	{attribute 'TcIecLibraryType'}
	{attribute 'external_name' := 'F_VN_ApplyYAxisInversionToAffineTransformationExp_GUID_95763161_5894_2E34_6A2A_637EF808A786'}
	(* Apply an inversion of the y-axis direction to an existing 2D affine transformation matrix. (expert function) *)
	FUNCTION F_VN_ApplyYAxisInversionToAffineTransformationExp : HRESULT
	VAR_IN_OUT
		aTransformationMatrix	:	TcVnMatrix2x3_LREAL;	(* Affine transformation matrix to which the inversion of the y-axis direction is applied *)
	END_VAR
	VAR_INPUT
		bUsePreMultiplication	:	BOOL;	(* Select if pre- or post-multiplication should be used *)
		hrPrev	:	HRESULT;	(* HRESULT indicating the result of previous operations (If SUCCEEDED(hrPrev) equals false, no operation is executed.) *)
	END_VAR

END_FUNCTION

// Functions/Geometric and Coordinate Transformations/F_VN_ConvertCartesianToPolarAngleImage

	{attribute 'TcIecLibraryType'}
	{attribute 'external_name' := 'F_VN_ConvertCartesianToPolarAngleImage_GUID_8785DF50_8290_2A16_55B0_D427D2D5A086'}
	(* Converts cartesian coordinates (x, y) to polar angle. *)
	FUNCTION F_VN_ConvertCartesianToPolarAngleImage : HRESULT
	VAR_INPUT
		ipSrcImageX	:	ITcVnImage;	(* Source image containing the x values (elements of type REAL or LREAL) *)
		ipSrcImageY	:	ITcVnImage;	(* Source image containing the y values (Same element type as ipSrcImageX) *)
		ipDestImageAng	:	REFERENCE TO ITcVnImage;	(* Destination image containing the angles (Same element type as source images. An appropriate destination image will be created if required.) *)
		hrPrev	:	HRESULT;	(* HRESULT indicating the result of previous operations (If SUCCEEDED(hrPrev) equals false, no operation is executed.) *)
	END_VAR

END_FUNCTION

// Functions/Geometric and Coordinate Transformations/F_VN_ConvertCartesianToPolarAngleImageExp

	{attribute 'TcIecLibraryType'}
	{attribute 'external_name' := 'F_VN_ConvertCartesianToPolarAngleImageExp_GUID_8D077096_5D1D_2FC1_51E8_F25300BF841D'}
	(* Converts cartesian coordinates (x, y) to polar angle. (expert function) *)
	FUNCTION F_VN_ConvertCartesianToPolarAngleImageExp : HRESULT
	VAR_INPUT
		ipSrcImageX	:	ITcVnImage;	(* Source image containing the x values (elements of type REAL or LREAL) *)
		ipSrcImageY	:	ITcVnImage;	(* Source image containing the y values (Same element type as ipSrcImageX) *)
		ipDestImageAng	:	REFERENCE TO ITcVnImage;	(* Destination image containing the angles (Same element type as source images. An appropriate destination image will be created if required.) *)
		bAngleInDegrees	:	BOOL;	(* Specifys, if the angles should be in degrees or radians *)
		hrPrev	:	HRESULT;	(* HRESULT indicating the result of previous operations (If SUCCEEDED(hrPrev) equals false, no operation is executed.) *)
	END_VAR

END_FUNCTION

// Functions/Geometric and Coordinate Transformations/F_VN_ConvertCartesianToPolarAngles

	{attribute 'TcIecLibraryType'}
	{attribute 'external_name' := 'F_VN_ConvertCartesianToPolarAngles_GUID_777B4F5A_64D8_2B5B_6D5A_3B670B4891DC'}
	(* Converts cartesian coordinates (x, y) to polar angle. *)
	FUNCTION F_VN_ConvertCartesianToPolarAngles : HRESULT
	VAR_INPUT
		ipSrcPointsCart	:	ITcVnContainer;	(* Container with cartesian points (ContainerType_Vector_TcVnPoint2_DINT or ContainerType_Vector_TcVnPoint2_REAL or ContainerType_Vector_TcVnPoint2_LREAL) *)
		ipDestAngles	:	REFERENCE TO ITcVnContainer;	(* Returns a container which is filled with the angles (ContainerType_Vector_REAL, if source points are of type TcVnPoint2_DINT or TcVnPoint2_REAL; else ContainerType_Vector_LREAL. Non-zero interface pointers are reused.) *)
		hrPrev	:	HRESULT;	(* HRESULT indicating the result of previous operations (If SUCCEEDED(hrPrev) equals false, no operation is executed.) *)
	END_VAR

END_FUNCTION

// Functions/Geometric and Coordinate Transformations/F_VN_ConvertCartesianToPolarAnglesExp

	{attribute 'TcIecLibraryType'}
	{attribute 'external_name' := 'F_VN_ConvertCartesianToPolarAnglesExp_GUID_C17BBC53_AA08_2C58_6EA5_EB565B2A30B9'}
	(* Converts cartesian coordinates (x, y) to polar angle. (expert function) *)
	FUNCTION F_VN_ConvertCartesianToPolarAnglesExp : HRESULT
	VAR_INPUT
		ipSrcPointsCart	:	ITcVnContainer;	(* Container with cartesian points (ContainerType_Vector_TcVnPoint2_DINT or ContainerType_Vector_TcVnPoint2_REAL or ContainerType_Vector_TcVnPoint2_LREAL) *)
		ipDestAngles	:	REFERENCE TO ITcVnContainer;	(* Returns a container which is filled with the angles (ContainerType_Vector_REAL, if source points are of type TcVnPoint2_DINT or TcVnPoint2_REAL; else ContainerType_Vector_LREAL. Non-zero interface pointers are reused.) *)
		bAngleInDegrees	:	BOOL;	(* Specify, if the angles should be in degrees or radians *)
		hrPrev	:	HRESULT;	(* HRESULT indicating the result of previous operations (If SUCCEEDED(hrPrev) equals false, no operation is executed.) *)
	END_VAR

END_FUNCTION

// Functions/Geometric and Coordinate Transformations/F_VN_ConvertCartesianToPolarImages

	{attribute 'TcIecLibraryType'}
	{attribute 'external_name' := 'F_VN_ConvertCartesianToPolarImages_GUID_68D50C9F_CB61_2D1C_5256_8997FCBD3F82'}
	(* Converts cartesian coordinates (x, y) to polar coordinates (magnitude, angle). *)
	FUNCTION F_VN_ConvertCartesianToPolarImages : HRESULT
	VAR_INPUT
		ipSrcImageX	:	ITcVnImage;	(* Source image containing the x values (elements of type REAL or LREAL) *)
		ipSrcImageY	:	ITcVnImage;	(* Source image containing the y values (Same element type as ipSrcImageX) *)
		ipDestImageMag	:	REFERENCE TO ITcVnImage;	(* Destination image containing the magnitudes (Same element type as source images. An appropriate destination image will be created if required.) *)
		ipDestImageAng	:	REFERENCE TO ITcVnImage;	(* Destination image containing the angles (Same element type as source images. An appropriate destination image will be created if required.) *)
		hrPrev	:	HRESULT;	(* HRESULT indicating the result of previous operations (If SUCCEEDED(hrPrev) equals false, no operation is executed.) *)
	END_VAR

END_FUNCTION

// Functions/Geometric and Coordinate Transformations/F_VN_ConvertCartesianToPolarImagesExp

	{attribute 'TcIecLibraryType'}
	{attribute 'external_name' := 'F_VN_ConvertCartesianToPolarImagesExp_GUID_57A46AC2_A055_2CB3_451E_4402032FA64B'}
	(* Converts cartesian coordinates (x, y) to polar coordinates (magnitude, angle). (expert function) *)
	FUNCTION F_VN_ConvertCartesianToPolarImagesExp : HRESULT
	VAR_INPUT
		ipSrcImageX	:	ITcVnImage;	(* Source image containing the x values (elements of type REAL or LREAL) *)
		ipSrcImageY	:	ITcVnImage;	(* Source image containing the y values (Same element type as ipSrcImageX) *)
		ipDestImageMag	:	REFERENCE TO ITcVnImage;	(* Destination image containing the magnitudes (Same element type as source images. An appropriate destination image will be created if required.) *)
		ipDestImageAng	:	REFERENCE TO ITcVnImage;	(* Destination image containing the angles (Same element type as source images. An appropriate destination image will be created if required.) *)
		bAngleInDegrees	:	BOOL;	(* Specifys, if the angles should be in degrees or radians *)
		hrPrev	:	HRESULT;	(* HRESULT indicating the result of previous operations (If SUCCEEDED(hrPrev) equals false, no operation is executed.) *)
	END_VAR

END_FUNCTION

// Functions/Geometric and Coordinate Transformations/F_VN_ConvertCartesianToPolarMagnitudeImage

	{attribute 'TcIecLibraryType'}
	{attribute 'external_name' := 'F_VN_ConvertCartesianToPolarMagnitudeImage_GUID_99EFD0C0_CF11_2C59_5201_85CBDF72A9FC'}
	(* Converts cartesian coordinates (x, y) to polar magnitude. *)
	FUNCTION F_VN_ConvertCartesianToPolarMagnitudeImage : HRESULT
	VAR_INPUT
		ipSrcImageX	:	ITcVnImage;	(* Source image containing the x values (elements of type REAL or LREAL) *)
		ipSrcImageY	:	ITcVnImage;	(* Source image containing the y values (Same element type as ipSrcImageX) *)
		ipDestImageMag	:	REFERENCE TO ITcVnImage;	(* Destination image containing the magnitudes (Same element type as source images. An appropriate destination image will be created if required.) *)
		hrPrev	:	HRESULT;	(* HRESULT indicating the result of previous operations (If SUCCEEDED(hrPrev) equals false, no operation is executed.) *)
	END_VAR

END_FUNCTION

// Functions/Geometric and Coordinate Transformations/F_VN_ConvertCartesianToPolarMagnitudes

	{attribute 'TcIecLibraryType'}
	{attribute 'external_name' := 'F_VN_ConvertCartesianToPolarMagnitudes_GUID_87575312_399C_21BE_5CEE_FFE66CC03CE2'}
	(* Converts cartesian coordinates (x, y) to polar magnitude. *)
	FUNCTION F_VN_ConvertCartesianToPolarMagnitudes : HRESULT
	VAR_INPUT
		ipSrcPointsCart	:	ITcVnContainer;	(* Container with cartesian points (ContainerType_Vector_TcVnPoint2_DINT or ContainerType_Vector_TcVnPoint2_REAL or ContainerType_Vector_TcVnPoint2_LREAL) *)
		ipDestMags	:	REFERENCE TO ITcVnContainer;	(* Returns a container which is filled with the magnitudes (ContainerType_Vector_REAL, if source points are of type TcVnPoint2_DINT or TcVnPoint2_REAL; else ContainerType_Vector_LREAL. Non-zero interface pointers are reused.) *)
		hrPrev	:	HRESULT;	(* HRESULT indicating the result of previous operations (If SUCCEEDED(hrPrev) equals false, no operation is executed.) *)
	END_VAR

END_FUNCTION

// Functions/Geometric and Coordinate Transformations/F_VN_ConvertCartesianToPolarPoints

	{attribute 'TcIecLibraryType'}
	{attribute 'external_name' := 'F_VN_ConvertCartesianToPolarPoints_GUID_8B11E781_4477_2A78_64E3_1080D7128B46'}
	(* Converts cartesian coordinates (x, y) to polar coordinates (magnitude, angle). *)
	FUNCTION F_VN_ConvertCartesianToPolarPoints : HRESULT
	VAR_INPUT
		ipSrcPointsCart	:	ITcVnContainer;	(* Container with cartesian points (ContainerType_Vector_TcVnPoint2_DINT or ContainerType_Vector_TcVnPoint2_REAL or ContainerType_Vector_TcVnPoint2_LREAL) *)
		ipDestPointsPolar	:	REFERENCE TO ITcVnContainer;	(* Returns a container which is filled with the converted points in polar coordinates (ContainerType_Vector_TcVnPoint2_REAL, if source points are of type TcVnPoint2_DINT or TcVnPoint2_REAL; else ContainerType_Vector_TcVnPoint2_LREAL. Non-zero interface pointers are reused.) *)
		hrPrev	:	HRESULT;	(* HRESULT indicating the result of previous operations (If SUCCEEDED(hrPrev) equals false, no operation is executed.) *)
	END_VAR

END_FUNCTION

// Functions/Geometric and Coordinate Transformations/F_VN_ConvertCartesianToPolarPointsExp

	{attribute 'TcIecLibraryType'}
	{attribute 'external_name' := 'F_VN_ConvertCartesianToPolarPointsExp_GUID_EBBE416A_22C1_27E0_4531_5F2A0458D967'}
	(* Converts cartesian coordinates (x, y) to polar coordinates (magnitude, angle). (expert function) *)
	FUNCTION F_VN_ConvertCartesianToPolarPointsExp : HRESULT
	VAR_INPUT
		ipSrcPointsCart	:	ITcVnContainer;	(* Container with cartesian points (ContainerType_Vector_TcVnPoint2_DINT or ContainerType_Vector_TcVnPoint2_REAL or ContainerType_Vector_TcVnPoint2_LREAL) *)
		ipDestPointsPolar	:	REFERENCE TO ITcVnContainer;	(* Returns a container which is filled with the converted points in polar coordinates (ContainerType_Vector_TcVnPoint2_REAL, if source points are of type TcVnPoint2_DINT or TcVnPoint2_REAL; else ContainerType_Vector_TcVnPoint2_LREAL. Non-zero interface pointers are reused.) *)
		bAngleInDegrees	:	BOOL;	(* Specifys, if the angles should be in degrees or radians *)
		hrPrev	:	HRESULT;	(* HRESULT indicating the result of previous operations (If SUCCEEDED(hrPrev) equals false, no operation is executed.) *)
	END_VAR

END_FUNCTION

// Functions/Geometric and Coordinate Transformations/F_VN_ConvertPolarToCartesianImages

	{attribute 'TcIecLibraryType'}
	{attribute 'external_name' := 'F_VN_ConvertPolarToCartesianImages_GUID_45E29034_812A_29F4_4EDE_5DEB6A02A42A'}
	(* Converts polar coordinates (magnitude, angle) to cartesian coordinates (x, y). *)
	FUNCTION F_VN_ConvertPolarToCartesianImages : HRESULT
	VAR_INPUT
		ipSrcImageMag	:	ITcVnImage;	(* Source image containing the magnitudes (elements of type REAL or LREAL) *)
		ipSrcImageAng	:	ITcVnImage;	(* Source image containing the angles (Same element type as ipSrcImageMag) *)
		ipDestImageX	:	REFERENCE TO ITcVnImage;	(* Destination image containing the x values (Same element type as source images. An appropriate destination image will be created if required.) *)
		ipDestImageY	:	REFERENCE TO ITcVnImage;	(* Destination image containing the y values (Same element type as source images. An appropriate destination image will be created if required.) *)
		hrPrev	:	HRESULT;	(* HRESULT indicating the result of previous operations (If SUCCEEDED(hrPrev) equals false, no operation is executed.) *)
	END_VAR

END_FUNCTION

// Functions/Geometric and Coordinate Transformations/F_VN_ConvertPolarToCartesianImagesExp

	{attribute 'TcIecLibraryType'}
	{attribute 'external_name' := 'F_VN_ConvertPolarToCartesianImagesExp_GUID_1AB5C748_33A4_22CB_7CB8_EEAC3F1ECB67'}
	(* Converts polar coordinates (magnitude, angle) to cartesian coordinates (x, y). (expert function) *)
	FUNCTION F_VN_ConvertPolarToCartesianImagesExp : HRESULT
	VAR_INPUT
		ipSrcImageMag	:	ITcVnImage;	(* Source image containing the magnitudes (elements of type REAL or LREAL) *)
		ipSrcImageAng	:	ITcVnImage;	(* Source image containing the angles (Same element type as ipSrcImageMag) *)
		ipDestImageX	:	REFERENCE TO ITcVnImage;	(* Destination image containing the x values (Same element type as source images. An appropriate destination image will be created if required.) *)
		ipDestImageY	:	REFERENCE TO ITcVnImage;	(* Destination image containing the y values (Same element type as source images. An appropriate destination image will be created if required.) *)
		bAngleInDegrees	:	BOOL;	(* Specifys, if the angles are in degrees or radians *)
		hrPrev	:	HRESULT;	(* HRESULT indicating the result of previous operations (If SUCCEEDED(hrPrev) equals false, no operation is executed.) *)
	END_VAR

END_FUNCTION

// Functions/Geometric and Coordinate Transformations/F_VN_ConvertPolarToCartesianPoints

	{attribute 'TcIecLibraryType'}
	{attribute 'external_name' := 'F_VN_ConvertPolarToCartesianPoints_GUID_CD991F11_BA52_23B9_7986_18C4D3FB967A'}
	(* Converts polar coordinates (magnitude, angle) to cartesian coordinates (x, y). *)
	FUNCTION F_VN_ConvertPolarToCartesianPoints : HRESULT
	VAR_INPUT
		ipSrcPointsPolar	:	ITcVnContainer;	(* Container with polar coordinates (ContainerType_Vector_TcVnPoint2_REAL or ContainerType_Vector_TcVnPoint2_LREAL) *)
		ipDestPointsCart	:	REFERENCE TO ITcVnContainer;	(* Returns a container which is filled with the converted points in cartesian coordinates (same type ID as ipSrcPointsPolar. Non-zero interface pointers are reused.) *)
		hrPrev	:	HRESULT;	(* HRESULT indicating the result of previous operations (If SUCCEEDED(hrPrev) equals false, no operation is executed.) *)
	END_VAR

END_FUNCTION

// Functions/Geometric and Coordinate Transformations/F_VN_ConvertPolarToCartesianPointsExp

	{attribute 'TcIecLibraryType'}
	{attribute 'external_name' := 'F_VN_ConvertPolarToCartesianPointsExp_GUID_918F4026_8031_2284_7371_9471AA009DB3'}
	(* Converts polar coordinates (magnitude, angle) to cartesian coordinates (x, y). (expert function) *)
	FUNCTION F_VN_ConvertPolarToCartesianPointsExp : HRESULT
	VAR_INPUT
		ipSrcPointsPolar	:	ITcVnContainer;	(* Container with polar coordinates (ContainerType_Vector_TcVnPoint2_REAL or ContainerType_Vector_TcVnPoint2_LREAL) *)
		ipDestPointsCart	:	REFERENCE TO ITcVnContainer;	(* Returns a container which is filled with the converted points in cartesian coordinates (same type ID as ipSrcPointsPolar. Non-zero interface pointers are reused.) *)
		bAngleInDegrees	:	BOOL;	(* Specifys, if the angles are in degrees or radians *)
		hrPrev	:	HRESULT;	(* HRESULT indicating the result of previous operations (If SUCCEEDED(hrPrev) equals false, no operation is executed.) *)
	END_VAR

END_FUNCTION

// Functions/Geometric and Coordinate Transformations/F_VN_DecomposeAffineTransformation

	{attribute 'TcIecLibraryType'}
	{attribute 'external_name' := 'F_VN_DecomposeAffineTransformation_GUID_98D5C342_86DD_2C0D_79C0_D5DCC34233C1'}
	(* Decompose an affine transformation matrix and return the rotation angle (clockwise) in radian. The decomposition method assumes the following order of transformation: Translation, Rotation, Scale, and Skew. *)
	FUNCTION F_VN_DecomposeAffineTransformation : HRESULT
	VAR_IN_OUT
		aAffineTransform	:	TcVnMatrix2x3_LREAL;	(* Affine transformation matrix *)
		fRotationAngle	:	LREAL;	(* Rotation angle (radian) in the clockwise direction. The rotation center is the origin point (0,0) *)
	END_VAR
	VAR_INPUT
		hrPrev	:	HRESULT;	(* HRESULT indicating the result of previous operations (If SUCCEEDED(hrPrev) equals false, no operation is executed.) *)
	END_VAR

END_FUNCTION

// Functions/Geometric and Coordinate Transformations/F_VN_DecomposeAffineTransformationExp

	{attribute 'TcIecLibraryType'}
	{attribute 'external_name' := 'F_VN_DecomposeAffineTransformationExp_GUID_9A76BFDE_9FD8_208E_5443_0689F70E8650'}
	(* Decompose an affine transformation matrix and return the rotation angle (clockwise) in radian, translation vector (pixels), scale, and skew vectors (angle in radian). The decomposition method assumes the following order of transformation: Translation, Rotation, Scale, and Skew. *)
	FUNCTION F_VN_DecomposeAffineTransformationExp : HRESULT
	VAR_IN_OUT
		aAffineTransform	:	TcVnMatrix2x3_LREAL;	(* Affine transformation matrix *)
		fRotationAngle	:	LREAL;	(* Rotation angle (radian) in the clockwise direction. The rotation center is the origin point (0,0) *)
		aTranslationVector	:	TcVnVector2_LREAL;	(* 2D translation vector. The values are in pixels *)
		aScaleVector	:	TcVnVector2_LREAL;	(* 2D scale vector  *)
		aSkewVector	:	TcVnVector2_LREAL;	(* 2D skew vector. The values are the skew angles in x and y directions in radian *)
	END_VAR
	VAR_INPUT
		hrPrev	:	HRESULT;	(* HRESULT indicating the result of previous operations (If SUCCEEDED(hrPrev) equals false, no operation is executed.) *)
	END_VAR

END_FUNCTION

// Functions/Geometric and Coordinate Transformations/F_VN_DecomposeHomography

	{attribute 'TcIecLibraryType'}
	{attribute 'external_name' := 'F_VN_DecomposeHomography_GUID_98F01A4A_1DBD_2075_5784_A350D33354E2'}
	(* Decompose a homography matrix into four solutions of rotation, translation, and plane normal. It returns two solutions (Ra, Ta, Nb) and (Rb, Tb, Nb). The third and the fourth solutions can be calculated as follows: (Ra, -Ta, -Na) and (Rb, -Tb, -Nb). *)
	FUNCTION F_VN_DecomposeHomography : HRESULT
	VAR_IN_OUT
		aHomography	:	TcVnMatrix3x3_LREAL;	(* Homography matrix (a perspective transformation between two planes) *)
		aCameraMatrix	:	TcVnMatrix3x3_LREAL;	(* Camera matrix *)
		aRotationMatrixA	:	TcVnMatrix3x3_LREAL;	(* Rotation matrix of the first solution (Ra) *)
		aTranslationVectorA	:	TcVnVector3_LREAL;	(* Translation vector of the first solution (Ta) *)
		aNormVectorA	:	TcVnVector3_LREAL;	(* Norm vector of the first solution (Na) *)
		aRotationMatrixB	:	TcVnMatrix3x3_LREAL;	(* Rotation matrix of the second solution (Rb) *)
		aTranslationVectorB	:	TcVnVector3_LREAL;	(* Translation vector of the second solution (Tb) *)
		aNormVectorB	:	TcVnVector3_LREAL;	(* Norm vector of the second solution Nb *)
	END_VAR
	VAR_INPUT
		hrPrev	:	HRESULT;	(* HRESULT indicating the result of previous operations (If SUCCEEDED(hrPrev) equals false, no operation is executed.) *)
	END_VAR
	VAR_OUTPUT
		nSolutions	:	UDINT;	(* Returns the number of solutions. In normal cases, it is equal four.  *)
	END_VAR

END_FUNCTION

// Functions/Geometric and Coordinate Transformations/F_VN_DecomposeHomographyExp

	{attribute 'TcIecLibraryType'}
	{attribute 'external_name' := 'F_VN_DecomposeHomographyExp_GUID_E4534782_F1E5_2C71_56D0_408A9351CD4C'}
	(* Decompose a homography matrix and verify four solutions of rotation, translation, and plane normal. It uses visible reference points being in front of the camera to confirm which solution(s) of the four solutions (maximum two solutions) are consistent with all reference points. *)
	FUNCTION F_VN_DecomposeHomographyExp : HRESULT
	VAR_IN_OUT
		aHomography	:	TcVnMatrix3x3_LREAL;	(* Homography matrix (a perspective transformation between two planes) *)
		aCameraMatrix	:	TcVnMatrix3x3_LREAL;	(* Camera matrix *)
		aRotationMatrixA	:	TcVnMatrix3x3_LREAL;	(* Rotation matrix of the first solution (Ra) *)
		aTranslationVectorA	:	TcVnVector3_LREAL;	(* Translation vector of the first solution (Ta) *)
		aNormVectorA	:	TcVnVector3_LREAL;	(* Norm vector of the first solution (Na) *)
		aRotationMatrixB	:	TcVnMatrix3x3_LREAL;	(* Rotation matrix of the second solution (Rb) *)
		aTranslationVectorB	:	TcVnVector3_LREAL;	(* Translation vector of the second solution (Tb) *)
		aNormVectorB	:	TcVnVector3_LREAL;	(* Norm vector of the second solution (Nb) *)
	END_VAR
	VAR_INPUT
		ipPointsSrc	:	ITcVnContainer;	(* Container with source points (ContainerType_Vector_TcVnPoint2_REAL) *)
		ipPointsDes	:	ITcVnContainer;	(* Container with destination points (same number as ipPoints1, ContainerType_Vector_TcVnPoint2_REAL) *)
		ipInlierMask	:	ITcVnContainer;	(* A mask marking the inliers (optional, set to 0 if not available; ContainerType_Vector_SINT or ContainerType_Vector_USINT) *)
		hrPrev	:	HRESULT;	(* HRESULT indicating the result of previous operations (If SUCCEEDED(hrPrev) equals false, no operation is executed.) *)
	END_VAR
	VAR_OUTPUT
		nSolutions	:	UDINT;	(* Return the number of true potential solutions [0,1, or 2].
							0: no true potential solutions for the given corresponding points are confirmed.
							1: the solution (Ra, Ta, Na) is confirmed.
							2: both solution (Ra, Ta, Na) and (Rb, Tb, Nb) are confirmed.
							In all cases the function returns two solutions (Ra, Ta, Nb) and (Rb, Tb, Nb). The third and the fourth solutions can be calculated as follows: (Ra, -Ta, -Na) and (Rb, -Tb, -Nb).
						 *)
	END_VAR

END_FUNCTION

// Functions/Geometric and Coordinate Transformations/F_VN_FlipImage

	{attribute 'TcIecLibraryType'}
	{attribute 'external_name' := 'F_VN_FlipImage_GUID_48B32E72_66CF_244B_574F_84B8CCCB3BE5'}
	(* Flip an image (mirror and shift back to prior coordinates). *)
	FUNCTION F_VN_FlipImage : HRESULT
	VAR_INPUT
		ipSrcImage	:	ITcVnImage;	(* Source image *)
		ipDestImage	:	REFERENCE TO ITcVnImage;	(* Destination image (An appropriate destination image will be created if required.) *)
		eFlipAxis	:	ETcVnFlipAxis;	(* Selects the axis around which to flip the image *)
		hrPrev	:	HRESULT;	(* HRESULT indicating the result of previous operations (If SUCCEEDED(hrPrev) equals false, no operation is executed.) *)
	END_VAR

END_FUNCTION

// Functions/Geometric and Coordinate Transformations/F_VN_GenerateAffineTransformationUnitMatrix2D

	{attribute 'TcIecLibraryType'}
	{attribute 'external_name' := 'F_VN_GenerateAffineTransformationUnitMatrix2D_GUID_0E766047_45D3_2A7A_5039_15231E2195FF'}
	(* Generate an affine transformation 2D unit matrix. *)
	FUNCTION F_VN_GenerateAffineTransformationUnitMatrix2D : HRESULT
	VAR_IN_OUT
		aTransformationMatrix	:	TcVnMatrix2x3_LREAL;	(* Resulting affine transformation unit matrix *)
	END_VAR
	VAR_INPUT
		hrPrev	:	HRESULT;	(* HRESULT indicating the result of previous operations (If SUCCEEDED(hrPrev) equals false, no operation is executed.) *)
	END_VAR

END_FUNCTION

// Functions/Geometric and Coordinate Transformations/F_VN_GetAffineTransformation

	{attribute 'TcIecLibraryType'}
	{attribute 'external_name' := 'F_VN_GetAffineTransformation_GUID_7F9475AC_C0C6_2ED5_5448_BF3DBD7E8953'}
	(* Calculate the affine transformation between three corresponding point pairs. The points mark the corners of the corresponding triangles. *)
	FUNCTION F_VN_GetAffineTransformation : HRESULT
	VAR_IN_OUT
		aSrcPoints	:	TcVnArray3_Point2_REAL;	(* Source points *)
		aDestPoints	:	TcVnArray3_Point2_REAL;	(* Destination points *)
		aTransformationMatrix	:	TcVnMatrix2x3_LREAL;	(* Resulting transformation matrix *)
	END_VAR
	VAR_INPUT
		hrPrev	:	HRESULT;	(* HRESULT indicating the result of previous operations (If SUCCEEDED(hrPrev) equals false, no operation is executed.) *)
	END_VAR

END_FUNCTION

// Functions/Geometric and Coordinate Transformations/F_VN_GetAffineTransformation2D

	{attribute 'TcIecLibraryType'}
	{attribute 'external_name' := 'F_VN_GetAffineTransformation2D_GUID_75CFB795_4F15_2741_5A15_1A9F0AAB074F'}
	(* Estimate the 2D affine transformation between two planar point sets using RANSAC algorithm. *)
	FUNCTION F_VN_GetAffineTransformation2D : HRESULT
	VAR_INPUT
		ipSrcPoints	:	ITcVnContainer;	(* Container with at least 3 source points (ContainerType_Vector_TcVnPoint2_REAL) *)
		ipDestPoints	:	ITcVnContainer;	(* Container with destination points (same number as ipSrcPoints, ContainerType_Vector_TcVnPoint2_REAL) *)
	END_VAR
	VAR_IN_OUT
		aAffineTransform	:	TcVnMatrix2x3_LREAL;	(* Returns the affine transformation matrix, which transforms the source points to the destination points *)
	END_VAR
	VAR_INPUT
		hrPrev	:	HRESULT;	(* HRESULT indicating the result of previous operations (If SUCCEEDED(hrPrev) equals false, no operation is executed.) *)
	END_VAR

END_FUNCTION

// Functions/Geometric and Coordinate Transformations/F_VN_GetAffineTransformation2DExp

	{attribute 'TcIecLibraryType'}
	{attribute 'external_name' := 'F_VN_GetAffineTransformation2DExp_GUID_A72EB0C5_44D0_245E_5406_EFAD4AF3D8CC'}
	(* Estimate the affine transformation between two planar point sets. (expert function) *)
	FUNCTION F_VN_GetAffineTransformation2DExp : HRESULT
	VAR_INPUT
		ipSrcPoints	:	ITcVnContainer;	(* Container with at least 3 source points (ContainerType_Vector_TcVnPoint2_REAL) *)
		ipDestPoints	:	ITcVnContainer;	(* Container with destination points (same number as ipSrcPoints, ContainerType_Vector_TcVnPoint2_REAL) *)
	END_VAR
	VAR_IN_OUT
		aAffineTransform	:	TcVnMatrix2x3_LREAL;	(* Returns the affine transformation matrix, which transforms the source points to the destination points *)
	END_VAR
	VAR_INPUT
		eAlgorithm	:	ETcVnEstimationAlgorithm;	(* Estimation algorithm (only RANSAC and LMEDS are supported) *)
		fReprojThreshold	:	LREAL;	(* Maximum allowed reprojection error to treat a point pair as an inlier *)
		ipInlierMask	:	REFERENCE TO ITcVnContainer;	(* Returns a mask marking the inliers (optional, set to 0 if not required; ContainerType_Vector_USINT) *)
		nMaxIterations	:	UDINT;	(* Maximum number of iterations *)
		fConfidence	:	LREAL;	(* Confidence (0..1) *)
		nRefineIters	:	UDINT;	(* Maximum number of iterations of Levenberg-Marquardt algorithm to refine further the affine transform (using only inliers). Set to 0 to disable refining. *)
		hrPrev	:	HRESULT;	(* HRESULT indicating the result of previous operations (If SUCCEEDED(hrPrev) equals false, no operation is executed.) *)
	END_VAR

END_FUNCTION

// Functions/Geometric and Coordinate Transformations/F_VN_GetPerspectiveTransformation

	{attribute 'TcIecLibraryType'}
	{attribute 'external_name' := 'F_VN_GetPerspectiveTransformation_GUID_F37A28EB_B072_2EC2_73AC_6B19B9A31E9E'}
	(* Calculate the perspective transformation between four corresponding point pairs. The points mark the corners of the corresponding rectangles. *)
	FUNCTION F_VN_GetPerspectiveTransformation : HRESULT
	VAR_IN_OUT
		aSrcPoints	:	TcVnArray4_Point2_REAL;	(* Source points *)
		aDestPoints	:	TcVnArray4_Point2_REAL;	(* Destination points *)
		aTransformationMatrix	:	TcVnMatrix3x3_LREAL;	(* Resulting transformation matrix *)
	END_VAR
	VAR_INPUT
		hrPrev	:	HRESULT;	(* HRESULT indicating the result of previous operations (If SUCCEEDED(hrPrev) equals false, no operation is executed.) *)
	END_VAR

END_FUNCTION

// Functions/Geometric and Coordinate Transformations/F_VN_Homography

	{attribute 'TcIecLibraryType'}
	{attribute 'external_name' := 'F_VN_Homography_GUID_8DBA4BBF_8913_20A2_43C2_DD73C62F3751'}
	(* Find the homography (perspective transformation) between two planar point sets using RANSAC algorithm. *)
	FUNCTION F_VN_Homography : HRESULT
	VAR_INPUT
		ipSrcPoints	:	ITcVnContainer;	(* Container with at least 4 source points (ContainerType_Vector_TcVnPoint2_REAL) *)
		ipDestPoints	:	ITcVnContainer;	(* Container with destination points (same number as ipSrcPoints, ContainerType_Vector_TcVnPoint2_REAL) *)
	END_VAR
	VAR_IN_OUT
		aPerspectiveTransform	:	TcVnMatrix3x3_LREAL;	(* Returns the perspective transformation matrix, which transforms the source points to the destination points *)
	END_VAR
	VAR_INPUT
		hrPrev	:	HRESULT;	(* HRESULT indicating the result of previous operations (If SUCCEEDED(hrPrev) equals false, no operation is executed.) *)
	END_VAR

END_FUNCTION

// Functions/Geometric and Coordinate Transformations/F_VN_HomographyExp

	{attribute 'TcIecLibraryType'}
	{attribute 'external_name' := 'F_VN_HomographyExp_GUID_A20F5D15_5E6B_2160_7CB0_9957C05F3906'}
	(* Find the homography (perspective transformation) between two planar point sets. (expert function) *)
	FUNCTION F_VN_HomographyExp : HRESULT
	VAR_INPUT
		ipSrcPoints	:	ITcVnContainer;	(* Container with at least 4 source points (ContainerType_Vector_TcVnPoint2_REAL) *)
		ipDestPoints	:	ITcVnContainer;	(* Container with destination points (same number as ipSrcPoints, ContainerType_Vector_TcVnPoint2_REAL) *)
	END_VAR
	VAR_IN_OUT
		aPerspectiveTransform	:	TcVnMatrix3x3_LREAL;	(* Returns the perspective transformation matrix, which transforms the source points to the destination points *)
	END_VAR
	VAR_INPUT
		eAlgorithm	:	ETcVnEstimationAlgorithm;	(* Estimation algorithm *)
		fReprojThreshold	:	LREAL;	(* Maximum allowed reprojection error to treat a point pair as an inlier (only for RANSAC, RHO) *)
		ipInlierMask	:	REFERENCE TO ITcVnContainer;	(* Returns a mask marking the inliers (optional, set to 0 if not required; ContainerType_Vector_SINT; only for RANSAC, LMEDS) *)
		nMaxIterations	:	UDINT;	(* Maximum number of RANSAC iterations *)
		fConfidence	:	LREAL;	(* Confidence (0..1) *)
		hrPrev	:	HRESULT;	(* HRESULT indicating the result of previous operations (If SUCCEEDED(hrPrev) equals false, no operation is executed.) *)
	END_VAR

END_FUNCTION

// Functions/Geometric and Coordinate Transformations/F_VN_InvertAffineTransformation

	{attribute 'TcIecLibraryType'}
	{attribute 'external_name' := 'F_VN_InvertAffineTransformation_GUID_ABA7A9B0_889B_28D8_73E4_DED30EBF1489'}
	(* Invert a 2D affine transformation matrix. The inverted transformation compensates the affine transformation on an image if it is used in the F_VN_WarpAffine function. *)
	FUNCTION F_VN_InvertAffineTransformation : HRESULT
	VAR_IN_OUT
		aTransformationMatrix	:	TcVnMatrix2x3_LREAL;	(* Source affine transformation matrix *)
		aInvertedTransformationMatrix	:	TcVnMatrix2x3_LREAL;	(* Resulting inverted affine transformation matrix *)
	END_VAR
	VAR_INPUT
		hrPrev	:	HRESULT;	(* HRESULT indicating the result of previous operations (If SUCCEEDED(hrPrev) equals false, no operation is executed.) *)
	END_VAR

END_FUNCTION

// Functions/Geometric and Coordinate Transformations/F_VN_WarpAffine

	{attribute 'TcIecLibraryType'}
	{attribute 'external_name' := 'F_VN_WarpAffine_GUID_10728BCD_6FE0_2CB9_535F_3F82DFB391B9'}
	(* Apply an affine transformation to an image. *)
	FUNCTION F_VN_WarpAffine : HRESULT
	VAR_INPUT
		ipSrcImage	:	ITcVnImage;	(* Source image *)
		ipDestImage	:	REFERENCE TO ITcVnImage;	(* Destination image (An appropriate image will be created if required.) *)
	END_VAR
	VAR_IN_OUT
		aTransformationMatrix	:	TcVnMatrix2x3_LREAL;	(* Affine transformation matrix *)
	END_VAR
	VAR_INPUT
		hrPrev	:	HRESULT;	(* HRESULT indicating the result of previous operations (If SUCCEEDED(hrPrev) equals false, no operation is executed.) *)
	END_VAR

END_FUNCTION

// Functions/Geometric and Coordinate Transformations/F_VN_PerspectiveTransformation

	{attribute 'TcIecLibraryType'}
	{attribute 'external_name' := 'F_VN_PerspectiveTransformation_GUID_967FB1A2_1C04_20ED_7F7A_354EA8433AB5'}
	(* Apply a perspective transformation (rotation + translation, e.g. from extrinsic calibration) to 3D point coordinates. *)
	FUNCTION F_VN_PerspectiveTransformation : HRESULT
	VAR_INPUT
		ipSrcPoints	:	ITcVnContainer;	(* Container with 3D source points (TcVnPoint3_REAL or TcVnPoint3_LREAL) *)
		ipDestPoints	:	REFERENCE TO ITcVnContainer;	(* Returns the transformed points (same type as ipSrcPoints) *)
	END_VAR
	VAR_IN_OUT
		aRotationMatrix	:	TcVnMatrix3x3_LREAL;	(* 3x3 rotation matrix *)
		aTranslationVector	:	TcVnVector3_LREAL;	(* Translation vector *)
	END_VAR
	VAR_INPUT
		hrPrev	:	HRESULT;	(* HRESULT indicating the result of previous operations (If SUCCEEDED(hrPrev) equals false, no operation is executed.) *)
	END_VAR

END_FUNCTION

// Functions/Geometric and Coordinate Transformations/F_VN_PyramidDown

	{attribute 'TcIecLibraryType'}
	{attribute 'external_name' := 'F_VN_PyramidDown_GUID_93185340_D05A_2222_621E_1414FDA6B37A'}
	(* Downsamples an image to half width and height. *)
	FUNCTION F_VN_PyramidDown : HRESULT
	VAR_INPUT
		ipSrcImage	:	ITcVnImage;	(* Source image *)
		ipDestImage	:	REFERENCE TO ITcVnImage;	(* Destination image (An appropriate destination image will be created if required.) *)
		hrPrev	:	HRESULT;	(* HRESULT indicating the result of previous operations (If SUCCEEDED(hrPrev) equals false, no operation is executed.) *)
	END_VAR

END_FUNCTION

// Functions/Geometric and Coordinate Transformations/F_VN_PyramidUp

	{attribute 'TcIecLibraryType'}
	{attribute 'external_name' := 'F_VN_PyramidUp_GUID_F01656A9_4836_2446_7AC7_A4904C8F1000'}
	(* Upsamples an image to double width and height. *)
	FUNCTION F_VN_PyramidUp : HRESULT
	VAR_INPUT
		ipSrcImage	:	ITcVnImage;	(* Source image *)
		ipDestImage	:	REFERENCE TO ITcVnImage;	(* Destination image (An appropriate destination image will be created if required.) *)
		hrPrev	:	HRESULT;	(* HRESULT indicating the result of previous operations (If SUCCEEDED(hrPrev) equals false, no operation is executed.) *)
	END_VAR

END_FUNCTION

// Functions/Geometric and Coordinate Transformations/F_VN_RemapImageToLogPolarSpace

	{attribute 'TcIecLibraryType'}
	{attribute 'external_name' := 'F_VN_RemapImageToLogPolarSpace_GUID_060AD528_6D67_2592_4F02_321CB9DA03A3'}
	(* Remap an image to log-polar space. *)
	FUNCTION F_VN_RemapImageToLogPolarSpace : HRESULT
	VAR_INPUT
		ipSrcImage	:	ITcVnImage;	(* Source image *)
		ipDestImage	:	REFERENCE TO ITcVnImage;	(* Destination image (Must not be the same as ipSrcImage! An appropriate destination image will be created if required.) *)
	END_VAR
	VAR_IN_OUT
		aCenter	:	TcVnPoint2_REAL;	(* Center point for the transformation *)
	END_VAR
	VAR_INPUT
		hrPrev	:	HRESULT;	(* HRESULT indicating the result of previous operations (If SUCCEEDED(hrPrev) equals false, no operation is executed.) *)
	END_VAR

END_FUNCTION

// Functions/Geometric and Coordinate Transformations/F_VN_RemapImageToLogPolarSpaceExp

	{attribute 'TcIecLibraryType'}
	{attribute 'external_name' := 'F_VN_RemapImageToLogPolarSpaceExp_GUID_F326A17F_212B_27D9_79D7_71DB73410236'}
	(* Remap an image to log-polar space. (expert function) *)
	FUNCTION F_VN_RemapImageToLogPolarSpaceExp : HRESULT
	VAR_INPUT
		ipSrcImage	:	ITcVnImage;	(* Source image *)
		ipDestImage	:	REFERENCE TO ITcVnImage;	(* Destination image (Must not be the same as ipSrcImage! An appropriate destination image will be created if required.) *)
	END_VAR
	VAR_IN_OUT
		aCenter	:	TcVnPoint2_REAL;	(* Center point for the transformation *)
	END_VAR
	VAR_INPUT
		fScale	:	LREAL;	(* Magnitude scale parameter, i.e. image width / ln(radius) (set to 0 for auto select) *)
		eInterpolationType	:	ETcVnInterpolationType;	(* Interpolation type *)
		hrPrev	:	HRESULT;	(* HRESULT indicating the result of previous operations (If SUCCEEDED(hrPrev) equals false, no operation is executed.) *)
	END_VAR

END_FUNCTION

// Functions/Geometric and Coordinate Transformations/F_VN_RemapImageToLogPolarSpaceExp2

	{attribute 'TcIecLibraryType'}
	{attribute 'external_name' := 'F_VN_RemapImageToLogPolarSpaceExp2_GUID_BBD4ED49_8137_2278_5B0B_EE05A71DE469'}
	(* Remap an image to log-polar space. (expert function) *)
	FUNCTION F_VN_RemapImageToLogPolarSpaceExp2 : HRESULT
	VAR_INPUT
		ipSrcImage	:	ITcVnImage;	(* Source image *)
		ipDestImage	:	REFERENCE TO ITcVnImage;	(* Destination image (Must not be the same as ipSrcImage! An appropriate destination image will be created if required.) *)
	END_VAR
	VAR_IN_OUT
		aCenter	:	TcVnPoint2_REAL;	(* Center point for the transformation *)
	END_VAR
	VAR_INPUT
		fScale	:	LREAL;	(* Magnitude scale parameter, i.e. image width / ln(radius) (set to 0 for auto select) *)
		eInterpolationType	:	ETcVnInterpolationType;	(* Interpolation type *)
		nDestWidth	:	DINT;	(* Destination image width (set to -1 for source image width, 0 to auto scale to transformed radius, > 0 for a user defined width) *)
		nDestHeight	:	DINT;	(* destination image height (set to -1 for source image height, 0 to auto scale to transformed radius * PI, > 0 for a user defined height) *)
		hrPrev	:	HRESULT;	(* HRESULT indicating the result of previous operations (If SUCCEEDED(hrPrev) equals false, no operation is executed.) *)
	END_VAR

END_FUNCTION

// Functions/Geometric and Coordinate Transformations/F_VN_RemapImageToPolarSpace

	{attribute 'TcIecLibraryType'}
	{attribute 'external_name' := 'F_VN_RemapImageToPolarSpace_GUID_B6D6ACB5_648A_2ECB_4E1F_2C85A691D8BD'}
	(* Remap an image to polar space. *)
	FUNCTION F_VN_RemapImageToPolarSpace : HRESULT
	VAR_INPUT
		ipSrcImage	:	ITcVnImage;	(* Source image *)
		ipDestImage	:	REFERENCE TO ITcVnImage;	(* Destination image (Must not be the same as ipSrcImage! An appropriate destination image will be created if required.) *)
	END_VAR
	VAR_IN_OUT
		aCenter	:	TcVnPoint2_REAL;	(* Center point for the transformation *)
	END_VAR
	VAR_INPUT
		hrPrev	:	HRESULT;	(* HRESULT indicating the result of previous operations (If SUCCEEDED(hrPrev) equals false, no operation is executed.) *)
	END_VAR

END_FUNCTION

// Functions/Geometric and Coordinate Transformations/F_VN_RemapImageToPolarSpaceExp

	{attribute 'TcIecLibraryType'}
	{attribute 'external_name' := 'F_VN_RemapImageToPolarSpaceExp_GUID_F0F3B1F8_3DBD_27FF_53C4_3ED8504E9F92'}
	(* Remap an image to polar space. (expert function) *)
	FUNCTION F_VN_RemapImageToPolarSpaceExp : HRESULT
	VAR_INPUT
		ipSrcImage	:	ITcVnImage;	(* Source image *)
		ipDestImage	:	REFERENCE TO ITcVnImage;	(* Destination image (Must not be the same as ipSrcImage! An appropriate destination image will be created if required.) *)
	END_VAR
	VAR_IN_OUT
		aCenter	:	TcVnPoint2_REAL;	(* Center point for the transformation *)
	END_VAR
	VAR_INPUT
		fMaxRadius	:	LREAL;	(* Maximum radius for the transformation (set to 0 for auto select) *)
		eInterpolationType	:	ETcVnInterpolationType;	(* Interpolation type *)
		hrPrev	:	HRESULT;	(* HRESULT indicating the result of previous operations (If SUCCEEDED(hrPrev) equals false, no operation is executed.) *)
	END_VAR

END_FUNCTION

// Functions/Geometric and Coordinate Transformations/F_VN_RemapImageToPolarSpaceExp2

	{attribute 'TcIecLibraryType'}
	{attribute 'external_name' := 'F_VN_RemapImageToPolarSpaceExp2_GUID_0B98FB53_46EB_2699_439F_D177142C2A0E'}
	(* Remap an image to polar space. (expert function) *)
	FUNCTION F_VN_RemapImageToPolarSpaceExp2 : HRESULT
	VAR_INPUT
		ipSrcImage	:	ITcVnImage;	(* Source image *)
		ipDestImage	:	REFERENCE TO ITcVnImage;	(* Destination image (Must not be the same as ipSrcImage! An appropriate destination image will be created if required.) *)
	END_VAR
	VAR_IN_OUT
		aCenter	:	TcVnPoint2_REAL;	(* Center point for the transformation *)
	END_VAR
	VAR_INPUT
		fMaxRadius	:	LREAL;	(* Maximum radius for the transformation (set to 0 for auto select) *)
		eInterpolationType	:	ETcVnInterpolationType;	(* Interpolation type *)
		nDestWidth	:	DINT;	(* Destination image width (set to -1 for source image width, 0 to auto scale to transformed radius, > 0 for a user defined width) *)
		nDestHeight	:	DINT;	(* destination image height (set to -1 for source image height, 0 to auto scale to transformed radius * PI, > 0 for a user defined height) *)
		hrPrev	:	HRESULT;	(* HRESULT indicating the result of previous operations (If SUCCEEDED(hrPrev) equals false, no operation is executed.) *)
	END_VAR

END_FUNCTION

// Functions/Geometric and Coordinate Transformations/F_VN_ResizeImage

	{attribute 'TcIecLibraryType'}
	{attribute 'external_name' := 'F_VN_ResizeImage_GUID_85E39FA5_3235_2B35_713A_6E9444FEE95F'}
	(* Resize an image using a specific interpolation type. *)
	FUNCTION F_VN_ResizeImage : HRESULT
	VAR_INPUT
		ipSrcImage	:	ITcVnImage;	(* Source image *)
		ipDestImage	:	REFERENCE TO ITcVnImage;	(* Destination image (An appropriate image will be created if required.) *)
		nWidth	:	UDINT;	(* New width *)
		nHeight	:	UDINT;	(* New height *)
		eInterpolationType	:	ETcVnInterpolationType;	(* Interpolation type *)
		hrPrev	:	HRESULT;	(* HRESULT indicating the result of previous operations (If SUCCEEDED(hrPrev) equals false, no operation is executed.) *)
	END_VAR

END_FUNCTION

// Functions/Geometric and Coordinate Transformations/F_VN_ResizeImageExp

	{attribute 'TcIecLibraryType'}
	{attribute 'external_name' := 'F_VN_ResizeImageExp_GUID_5FE45245_BBBE_2AAB_6763_04E36D61955B'}
	(* Resize an image using a specific interpolation type while maintaining its aspect ratio. (expert function) *)
	FUNCTION F_VN_ResizeImageExp : HRESULT
	VAR_INPUT
		ipSrcImage	:	ITcVnImage;	(* Source image *)
		ipDestImage	:	REFERENCE TO ITcVnImage;	(* Destination image (An appropriate image will be created if required.) *)
		nWidth	:	UDINT;	(* New width *)
		nHeight	:	UDINT;	(* New height *)
		eInterpolationType	:	ETcVnInterpolationType;	(* Interpolation type *)
		ePaddingMode	:	ETcVnPaddingMode;	(* Image padding mode *)
	END_VAR
	VAR_IN_OUT
		aBorderValue	:	TcVnVector4_LREAL;	(* Border value, if TCVN_PM_LETTERBOX is used *)
	END_VAR
	VAR_INPUT
		hrPrev	:	HRESULT;	(* HRESULT indicating the result of previous operations (If SUCCEEDED(hrPrev) equals false, no operation is executed.) *)
	END_VAR

END_FUNCTION

// Functions/Geometric and Coordinate Transformations/F_VN_RotateImage

	{attribute 'TcIecLibraryType'}
	{attribute 'external_name' := 'F_VN_RotateImage_GUID_E4386E12_392F_2B14_5E06_302D07DFCCA2'}
	(* Rotate an image by 90, 180, or 270 degrees in clockwise direction. *)
	FUNCTION F_VN_RotateImage : HRESULT
	VAR_INPUT
		ipSrcImage	:	ITcVnImage;	(* Source image *)
		ipDestImage	:	REFERENCE TO ITcVnImage;	(* Destination image (An appropriate image will be created if required.) *)
		eAngle	:	ETcVnRotationAngle;	(* Rotation angle *)
		hrPrev	:	HRESULT;	(* HRESULT indicating the result of previous operations (If SUCCEEDED(hrPrev) equals false, no operation is executed.) *)
	END_VAR

END_FUNCTION

// Functions/Geometric and Coordinate Transformations/F_VN_RotateImageExp

	{attribute 'TcIecLibraryType'}
	{attribute 'external_name' := 'F_VN_RotateImageExp_GUID_CAB32E81_B9B8_2C36_6744_1F946B8D5FF9'}
	(* Rotate an image by an individual rotation angle in degrees. *)
	FUNCTION F_VN_RotateImageExp : HRESULT
	VAR_INPUT
		ipSrcImage	:	ITcVnImage;	(* Source image *)
		ipDestImage	:	REFERENCE TO ITcVnImage;	(* Destination image (An appropriate image will be created if required.) *)
		fAngleDeg	:	LREAL;	(* Rotation angle in degree (positive: counter-clockwise, negative: clockwise) *)
		bAdjustDestSize	:	BOOL;	(* If true, ipDestImage size is adjusted so that the whole rotated ipSrcImage is contained. Otherwise, ipDestImage size is set to ipSrcImage size. *)
		hrPrev	:	HRESULT;	(* HRESULT indicating the result of previous operations (If SUCCEEDED(hrPrev) equals false, no operation is executed.) *)
	END_VAR

END_FUNCTION

// Functions/Geometric and Coordinate Transformations/F_VN_RotateImageExp2

	{attribute 'TcIecLibraryType'}
	{attribute 'external_name' := 'F_VN_RotateImageExp2_GUID_ED649F8E_1AFF_2675_6CD5_0E2314288623'}
	(* Rotate an image by an individual rotation angle in degrees. (expert function) *)
	FUNCTION F_VN_RotateImageExp2 : HRESULT
	VAR_INPUT
		ipSrcImage	:	ITcVnImage;	(* Source image *)
		ipDestImage	:	REFERENCE TO ITcVnImage;	(* Destination image (An appropriate image will be created if required.) *)
		fAngleDeg	:	LREAL;	(* Rotation angle in degree (positive: counter-clockwise, negative: clockwise) *)
		bAdjustDestSize	:	BOOL;	(* If true, ipDestImage size is adjusted so that the whole rotated ipSrcImage is contained. Otherwise, ipDestImage size is set to ipSrcImage size. *)
		eInterpolationType	:	ETcVnInterpolationType;	(* Interpolation method *)
		eBorderInterpolation	:	ETcVnBorderInterpolationMethod;	(* Border interpolation method (ISOLATED not supported) *)
	END_VAR
	VAR_IN_OUT
		aBorderValue	:	TcVnVector4_LREAL;	(* Border value, if CONSTANT is used *)
	END_VAR
	VAR_INPUT
		hrPrev	:	HRESULT;	(* HRESULT indicating the result of previous operations (If SUCCEEDED(hrPrev) equals false, no operation is executed.) *)
	END_VAR

END_FUNCTION

// Functions/Geometric and Coordinate Transformations/F_VN_WarpAffineExp

	{attribute 'TcIecLibraryType'}
	{attribute 'external_name' := 'F_VN_WarpAffineExp_GUID_8D589228_A9C5_2069_47F9_FA5ED2CBEA6C'}
	(* Apply an affine transformation to an image. (expert function) *)
	FUNCTION F_VN_WarpAffineExp : HRESULT
	VAR_INPUT
		ipSrcImage	:	ITcVnImage;	(* Source image *)
		ipDestImage	:	REFERENCE TO ITcVnImage;	(* Destination image (An appropriate image will be created if required.) *)
	END_VAR
	VAR_IN_OUT
		aTransformationMatrix	:	TcVnMatrix2x3_LREAL;	(* Affine transformation matrix *)
	END_VAR
	VAR_INPUT
		nDestWidth	:	UDINT;	(* Width of the destination image *)
		nDestHeight	:	UDINT;	(* Height of the destination image *)
		eInterpolationType	:	ETcVnInterpolationType;	(* Interpolation method *)
		bWarpInverse	:	BOOL;	(* Handle aTransformationMatrix as the inverse transformation *)
		eBorderInterpolation	:	ETcVnBorderInterpolationMethod;	(* Border interpolation method (ISOLATED not supported) *)
		fBorderValue	:	LREAL;	(* Border value, if CONSTANT is used *)
		hrPrev	:	HRESULT;	(* HRESULT indicating the result of previous operations (If SUCCEEDED(hrPrev) equals false, no operation is executed.) *)
	END_VAR

END_FUNCTION

// Functions/Geometric and Coordinate Transformations/F_VN_WarpAffine_Container

	{attribute 'TcIecLibraryType'}
	{attribute 'external_name' := 'F_VN_WarpAffine_Container_GUID_D5318516_D2B2_22D4_7205_75520F626C63'}
	(* Apply an affine transformation to a container of 2D points. *)
	FUNCTION F_VN_WarpAffine_Container : HRESULT
	VAR_INPUT
		ipSrcPoints	:	ITcVnContainer;	(* Source points (ContainerType_Vector_TcVnPoint2_DINT or ContainerType_Vector_TcVnPoint2_REAL or ContainerType_Vector_TcVnPoint2_LREAL) *)
		ipDestPoints	:	REFERENCE TO ITcVnContainer;	(* Returns the transformed points (same type ID as ipSrcPoints; Non-zero interface pointers are reused.) *)
	END_VAR
	VAR_IN_OUT
		aTransformationMatrix	:	TcVnMatrix2x3_LREAL;	(* Affine transformation matrix *)
	END_VAR
	VAR_INPUT
		hrPrev	:	HRESULT;	(* HRESULT indicating the result of previous operations (If SUCCEEDED(hrPrev) equals false, no operation is executed.) *)
	END_VAR

END_FUNCTION

// Functions/Geometric and Coordinate Transformations/F_VN_WarpAffine_Point

	{attribute 'TcIecLibraryType'}
	{attribute 'external_name' := 'F_VN_WarpAffine_Point_GUID_64F6FA36_EEA9_27AC_4E70_B4598808BC31'}
	(* Apply an affine transformation to a 2D point. *)
	FUNCTION F_VN_WarpAffine_Point : HRESULT
	VAR_IN_OUT
		aSrcPoint	:	TcVnPoint2_LREAL;	(* Source point *)
		aDestPoint	:	TcVnPoint2_LREAL;	(* Destination point *)
		aTransformationMatrix	:	TcVnMatrix2x3_LREAL;	(* Affine transformation matrix *)
	END_VAR
	VAR_INPUT
		hrPrev	:	HRESULT;	(* HRESULT indicating the result of previous operations (If SUCCEEDED(hrPrev) equals false, no operation is executed.) *)
	END_VAR

END_FUNCTION

// Functions/Geometric and Coordinate Transformations/F_VN_WarpAffine_Rectangle

	{attribute 'TcIecLibraryType'}
	{attribute 'external_name' := 'F_VN_WarpAffine_Rectangle_GUID_349E786A_A3E2_24DF_496F_99B2F0AD41C8'}
	(* Use an affine transform to warp a rectangle. *)
	FUNCTION F_VN_WarpAffine_Rectangle : HRESULT
	VAR_INPUT
		nTopLeftX	:	UDINT;	(* x coordinate of the top left corner *)
		nTopLeftY	:	UDINT;	(* y coordinate of the top left corner *)
		nBottomRightX	:	UDINT;	(* x coordinate of the bottom right corner *)
		nBottomRightY	:	UDINT;	(* y coordinate of the bottom right corner *)
		ipDestPoints	:	REFERENCE TO ITcVnContainer;	(* Returns the 4 transformed points (ContainerType_Vector_TcVnPoint2_REAL) *)
	END_VAR
	VAR_IN_OUT
		aTransformationMatrix	:	TcVnMatrix2x3_LREAL;	(* Affine transformation matrix *)
	END_VAR
	VAR_INPUT
		hrPrev	:	HRESULT;	(* HRESULT indicating the result of previous operations (If SUCCEEDED(hrPrev) equals false, no operation is executed.) *)
	END_VAR

END_FUNCTION

// Functions/Geometric and Coordinate Transformations/F_VN_WarpPerspective

	{attribute 'TcIecLibraryType'}
	{attribute 'external_name' := 'F_VN_WarpPerspective_GUID_92C4C697_D96A_21A3_5E0B_43BF2E689690'}
	(* Apply a perspective transformation to an image. *)
	FUNCTION F_VN_WarpPerspective : HRESULT
	VAR_INPUT
		ipSrcImage	:	ITcVnImage;	(* Source image *)
		ipDestImage	:	REFERENCE TO ITcVnImage;	(* Destination image (An appropriate image will be created if required.) *)
	END_VAR
	VAR_IN_OUT
		aTransformationMatrix	:	TcVnMatrix3x3_LREAL;	(* Perspective transformation matrix *)
	END_VAR
	VAR_INPUT
		hrPrev	:	HRESULT;	(* HRESULT indicating the result of previous operations (If SUCCEEDED(hrPrev) equals false, no operation is executed.) *)
	END_VAR

END_FUNCTION

// Functions/Geometric and Coordinate Transformations/F_VN_WarpPerspective_Container

	{attribute 'TcIecLibraryType'}
	{attribute 'external_name' := 'F_VN_WarpPerspective_Container_GUID_9911AD13_FEFC_2E53_7837_1268CAC6BE72'}
	(* Apply a perspective transformation to a container of 2D points. *)
	FUNCTION F_VN_WarpPerspective_Container : HRESULT
	VAR_INPUT
		ipSrcPoints	:	ITcVnContainer;	(* Source points (ContainerType_Vector_TcVnPoint2_DINT or ContainerType_Vector_TcVnPoint2_REAL or ContainerType_Vector_TcVnPoint2_LREAL) *)
		ipDestPoints	:	REFERENCE TO ITcVnContainer;	(* Returns the transformed points (same type ID as ipSrcPoints; Non-zero interface pointers are reused.) *)
	END_VAR
	VAR_IN_OUT
		aTransformationMatrix	:	TcVnMatrix3x3_LREAL;	(* Perspective transformation matrix *)
	END_VAR
	VAR_INPUT
		hrPrev	:	HRESULT;	(* HRESULT indicating the result of previous operations (If SUCCEEDED(hrPrev) equals false, no operation is executed.) *)
	END_VAR

END_FUNCTION

// Functions/Geometric and Coordinate Transformations/F_VN_WarpPerspectiveExp

	{attribute 'TcIecLibraryType'}
	{attribute 'external_name' := 'F_VN_WarpPerspectiveExp_GUID_6992E43D_094C_24B6_4B42_8C5044278B7E'}
	(* Apply a perspective transformation to an image. (expert function) *)
	FUNCTION F_VN_WarpPerspectiveExp : HRESULT
	VAR_INPUT
		ipSrcImage	:	ITcVnImage;	(* Source image *)
		ipDestImage	:	REFERENCE TO ITcVnImage;	(* Destination image (An appropriate image will be created if required.) *)
	END_VAR
	VAR_IN_OUT
		aTransformationMatrix	:	TcVnMatrix3x3_LREAL;	(* Perspective transformation matrix *)
	END_VAR
	VAR_INPUT
		nDestWidth	:	UDINT;	(* Width of the destination image *)
		nDestHeight	:	UDINT;	(* Height of the destination image *)
		eInterpolationType	:	ETcVnInterpolationType;	(* Interpolation method *)
		bWarpInverse	:	BOOL;	(* Handle aTransformationMatrix as the inverse transformation *)
		eBorderInterpolation	:	ETcVnBorderInterpolationMethod;	(* Border interpolation method (ISOLATED not supported) *)
		fBorderValue	:	LREAL;	(* Border value, if CONSTANT is used *)
		hrPrev	:	HRESULT;	(* HRESULT indicating the result of previous operations (If SUCCEEDED(hrPrev) equals false, no operation is executed.) *)
	END_VAR

END_FUNCTION

// Functions/Geometric and Coordinate Transformations/F_VN_WarpPerspective_Point

	{attribute 'TcIecLibraryType'}
	{attribute 'external_name' := 'F_VN_WarpPerspective_Point_GUID_624CDB7B_2111_2615_5471_76DD46E827B8'}
	(* Apply a perspective transformation to a 2D point. *)
	FUNCTION F_VN_WarpPerspective_Point : HRESULT
	VAR_IN_OUT
		aSrcPoint	:	TcVnPoint2_LREAL;	(* Source point *)
		aDestPoint	:	TcVnPoint2_LREAL;	(* Destination point *)
		aTransformationMatrix	:	TcVnMatrix3x3_LREAL;	(* Perspective transformation matrix *)
	END_VAR
	VAR_INPUT
		hrPrev	:	HRESULT;	(* HRESULT indicating the result of previous operations (If SUCCEEDED(hrPrev) equals false, no operation is executed.) *)
	END_VAR

END_FUNCTION

// Functions/Geometric and Coordinate Transformations/F_VN_WarpPerspective_Rectangle

	{attribute 'TcIecLibraryType'}
	{attribute 'external_name' := 'F_VN_WarpPerspective_Rectangle_GUID_9421E5F0_C129_222F_4FD2_3B5FE8634611'}
	(* Use a perspective transform to warp a rectangle. *)
	FUNCTION F_VN_WarpPerspective_Rectangle : HRESULT
	VAR_INPUT
		nTopLeftX	:	UDINT;	(* x coordinate of the top left corner *)
		nTopLeftY	:	UDINT;	(* y coordinate of the top left corner *)
		nBottomRightX	:	UDINT;	(* x coordinate of the bottom right corner *)
		nBottomRightY	:	UDINT;	(* y coordinate of the bottom right corner *)
		ipDestPoints	:	REFERENCE TO ITcVnContainer;	(* Returns the 4 transformed points (ContainerType_Vector_TcVnPoint2_REAL) *)
	END_VAR
	VAR_IN_OUT
		aTransformationMatrix	:	TcVnMatrix3x3_LREAL;	(* Perspective transformation matrix *)
	END_VAR
	VAR_INPUT
		hrPrev	:	HRESULT;	(* HRESULT indicating the result of previous operations (If SUCCEEDED(hrPrev) equals false, no operation is executed.) *)
	END_VAR

END_FUNCTION

// Functions/Image Color and Contrast Processing/F_VN_ApplyColorMap

	{attribute 'TcIecLibraryType'}
	{attribute 'external_name' := 'F_VN_ApplyColorMap_GUID_02E02083_2ADA_2330_5620_DC49DF11C979'}
	(* Apply a color map to a gray-level image. *)
	FUNCTION F_VN_ApplyColorMap : HRESULT
	VAR_INPUT
		ipSrcImage	:	ITcVnImage;	(* Source image (TCVN_ET_USINT or TCVN_ET_UINT, 1 channel) *)
		ipDestImage	:	REFERENCE TO ITcVnImage;	(* Returns the colored image (TCVN_ET_USINT, 3 channel. An appropriate image will be created if required.) *)
		ipColorMap	:	ITcVnContainer;	(* Color map to be applied to ipSrcImage (ContainerType_Vector_TcVnVector3_REAL with 256 or 65536 elements, dependent on ipSrcImage type). Can be either custom or created with F_VN_GenerateColorMap. *)
		hrPrev	:	HRESULT;	(* HRESULT indicating the result of previous operations (If SUCCEEDED(hrPrev) equals false, no operation is executed.) *)
	END_VAR

END_FUNCTION

// Functions/Image Color and Contrast Processing/F_VN_GenerateColorMap

	{attribute 'TcIecLibraryType'}
	{attribute 'external_name' := 'F_VN_GenerateColorMap_GUID_1C339FC3_131A_2A5F_7D73_ACDFC1E1D3FE'}
	(* Generates a pre-defined color map. *)
	FUNCTION F_VN_GenerateColorMap : HRESULT
	VAR_INPUT
		ipColorMap	:	REFERENCE TO ITcVnContainer;	(* Returns the color map (ContainerType_Vector_TcVnVector3_REAL with 256 or 65536 elements) *)
		eColorMap	:	ETcVnColorMap;	(* Selects a color map (similar to GNU Octave/MATLAB types) *)
		eColorMapSize	:	ETcVnColorMapSize;	(* Defines how many elements the generated color map should have *)
		hrPrev	:	HRESULT;	(* HRESULT indicating the result of previous operations (If SUCCEEDED(hrPrev) equals false, no operation is executed.) *)
	END_VAR

END_FUNCTION

// Functions/Image Color and Contrast Processing/F_VN_ApplyLut

	{attribute 'TcIecLibraryType'}
	{attribute 'external_name' := 'F_VN_ApplyLut_GUID_0052ADF5_B9C2_271B_59F0_B10945EEB867'}
	(* Apply a lookup table to an image to manipulate its colors. *)
	FUNCTION F_VN_ApplyLut : HRESULT
	VAR_INPUT
		ipSrcImage	:	ITcVnImage;	(* Source image (1-4 channels of 8 or 16 bit types SINT, USINT, INT, UINT) *)
		ipDestImage	:	REFERENCE TO ITcVnImage;	(* Returns the result image (same size, type and channels as ipSrcImage. An appropriate image will be created if required.) *)
		ipLut	:	ITcVnContainer;	(* Lookup table with elements matching ipSrcImage type and either 256 (8 bit images) or 65536 (16 bit images) elements. E.g. ContainerType_Vector_USINT for 1-4 channel USINT image (in this case, the same lookup values are used for each channel) or ContainerType_Vector_TcVnVector3_USINT for a 3 channel USINT image (in this case, each channel uses an individual lookup value).
						 *)
		hrPrev	:	HRESULT;	(* HRESULT indicating the result of previous operations (If SUCCEEDED(hrPrev) equals false, no operation is executed.) *)
	END_VAR

END_FUNCTION

// Functions/Image Color and Contrast Processing/F_VN_Clahe

	{attribute 'TcIecLibraryType'}
	{attribute 'external_name' := 'F_VN_Clahe_GUID_32B34DC5_63BF_2EBD_6EF8_A47D0973E1A9'}
	(* Apply Constrast Limited Adaptive Histogram Equalization. This applies local histogram equalization to individual tiles. *)
	FUNCTION F_VN_Clahe : HRESULT
	VAR_INPUT
		ipSrcImage	:	ITcVnImage;	(* Source image (TCVN_ET_USINT or TCVN_ET_UINT, 1 channel) *)
		ipDestImage	:	REFERENCE TO ITcVnImage;	(* Returns the resulting image (An appropriate image will be created if required.) *)
		hrPrev	:	HRESULT;	(* HRESULT indicating the result of previous operations (If SUCCEEDED(hrPrev) equals false, no operation is executed.) *)
	END_VAR

END_FUNCTION

// Functions/Image Color and Contrast Processing/F_VN_ClaheExp

	{attribute 'TcIecLibraryType'}
	{attribute 'external_name' := 'F_VN_ClaheExp_GUID_888F7867_0895_2EDB_5284_E45AE9AFB287'}
	(* Apply Constrast Limited Adaptive Histogram Equalization. This applies local histogram equalization to individual tiles. (expert function) *)
	FUNCTION F_VN_ClaheExp : HRESULT
	VAR_INPUT
		ipSrcImage	:	ITcVnImage;	(* Source image (TCVN_ET_USINT or TCVN_ET_UINT, 1 channel) *)
		ipDestImage	:	REFERENCE TO ITcVnImage;	(* Returns the resulting image (An appropriate image will be created if required.) *)
		fClipLimit	:	LREAL;	(* Threshold for contrast limit (set to <= 0 to disable clipping) *)
		nTilesX	:	UDINT;	(* Number of tiles in x direction *)
		nTilesY	:	UDINT;	(* Number of tiles in y direction *)
		hrPrev	:	HRESULT;	(* HRESULT indicating the result of previous operations (If SUCCEEDED(hrPrev) equals false, no operation is executed.) *)
	END_VAR

END_FUNCTION

// Functions/Image Color and Contrast Processing/F_VN_ConvertColorSpace

	{attribute 'TcIecLibraryType'}
	{attribute 'external_name' := 'F_VN_ConvertColorSpace_GUID_640938E6_2360_27C4_5A75_196D6D225F7D'}
	(* Convert image from one color space to another. *)
	FUNCTION F_VN_ConvertColorSpace : HRESULT
	VAR_INPUT
		ipSrcImage	:	ITcVnImage;	(* Source image *)
		ipDestImage	:	REFERENCE TO ITcVnImage;	(* Destination image (An appropriate destination image will be created if required.) *)
		eTransform	:	ETcVnColorSpaceTransform;	(* Transforms to be applied *)
		hrPrev	:	HRESULT;	(* HRESULT indicating the result of previous operations (If SUCCEEDED(hrPrev) equals false, no operation is executed.) *)
	END_VAR

END_FUNCTION

// Functions/Image Color and Contrast Processing/F_VN_GenerateCustomColorMap

	{attribute 'TcIecLibraryType'}
	{attribute 'external_name' := 'F_VN_GenerateCustomColorMap_GUID_7807816D_A877_2A75_6CEF_656260BAF6F9'}
	(* Generate a custom color map by interpolating between user defined colors (equally distributed, linear for each channel). *)
	FUNCTION F_VN_GenerateCustomColorMap : HRESULT
	VAR_INPUT
		ipColorMap	:	REFERENCE TO ITcVnContainer;	(* Returns the color map (ContainerType_Vector_TcVnVector3_REAL with 256 or 65536 elements) *)
		ipInitialColors	:	ITcVnContainer;	(* User defined colors (ContainerType_Vector_TcVnVector3_REAL, at least 2 elements) *)
		eColorMapSize	:	ETcVnColorMapSize;	(* Defines how many elements the generated color map should have *)
		hrPrev	:	HRESULT;	(* HRESULT indicating the result of previous operations (If SUCCEEDED(hrPrev) equals false, no operation is executed.) *)
	END_VAR

END_FUNCTION

// Functions/Image Color and Contrast Processing/F_VN_Histogram

	{attribute 'TcIecLibraryType'}
	{attribute 'external_name' := 'F_VN_Histogram_GUID_14467E81_0DA6_2ABB_4C47_752351FDB059'}
	(* Calculate the (multi-channel) histogram of an image. *)
	FUNCTION F_VN_Histogram : HRESULT
	VAR_INPUT
		ipSrcImage	:	ITcVnImage;	(* Source image *)
		ipDestHistogram	:	REFERENCE TO ITcVnContainer;	(* Returns a container with a multi-channel histogram, where every channel is represented as a vector of UDINT (ContainerType_Vector_Vector_UDINT. Non-zero interface pointers are reused.) *)
		hrPrev	:	HRESULT;	(* HRESULT indicating the result of previous operations (If SUCCEEDED(hrPrev) equals false, no operation is executed.) *)
	END_VAR

END_FUNCTION

// Functions/Image Color and Contrast Processing/F_VN_HistogramExp

	{attribute 'TcIecLibraryType'}
	{attribute 'external_name' := 'F_VN_HistogramExp_GUID_9F6C1F38_E3C9_2DCC_6A90_180641582A01'}
	(* Calculate the (multi-channel) histogram of an image. (expert function) *)
	FUNCTION F_VN_HistogramExp : HRESULT
	VAR_INPUT
		ipSrcImage	:	ITcVnImage;	(* Source image *)
		ipDestHistogram	:	REFERENCE TO ITcVnContainer;	(* Returns a container with a multi-channel histogram, where every channel is represented as a vector of UDINT (ContainerType_Vector_Vector_UDINT. Non-zero interface pointers are reused.) *)
	END_VAR
	VAR_IN_OUT
		nBins	:	UDINT;	(* Desired number of bins or 0 to keep the default for the corresponding image format (in) and default number of bins (out) *)
		fLowerBound	:	LREAL;	(* Lower (inclusive) boundary of the 0-th histogram bin (in), or receive the default if fLowerBound AND fUpperBound are set to 0 (out) *)
		fUpperBound	:	LREAL;	(* Upper (exclusive) boundary of the last histogram bin nBins-1 (in), or receive the default if fLowerBound AND fUpperBound are set to 0 (out) *)
	END_VAR
	VAR_INPUT
		ipMask	:	ITcVnImage;	(* Source image mask (TCVN_ET_USINT, 1 channel. Mask is optional, set to 0 if not required.) *)
		hrPrev	:	HRESULT;	(* HRESULT indicating the result of previous operations (If SUCCEEDED(hrPrev) equals false, no operation is executed.) *)
	END_VAR

END_FUNCTION

// Functions/Image Color and Contrast Processing/F_VN_HistogramEqualization

	{attribute 'TcIecLibraryType'}
	{attribute 'external_name' := 'F_VN_HistogramEqualization_GUID_B986CCF2_AF54_2F11_572B_95B27527F16C'}
	(* Equalize the histogram of a grayscale or rgb image, which normalizes the brightness and improves the contrast. *)
	FUNCTION F_VN_HistogramEqualization : HRESULT
	VAR_INPUT
		ipSrcImage	:	ITcVnImage;	(* Source image (USINT) *)
		ipDestImage	:	REFERENCE TO ITcVnImage;	(* Destination image (An appropriate destination image will be created if required.) *)
		hrPrev	:	HRESULT;	(* HRESULT indicating the result of previous operations (If SUCCEEDED(hrPrev) equals false, no operation is executed.) *)
	END_VAR

END_FUNCTION

// Functions/Image Color and Contrast Processing/F_VN_HistogramEqualizationExp

	{attribute 'TcIecLibraryType'}
	{attribute 'external_name' := 'F_VN_HistogramEqualizationExp_GUID_D39515B8_559F_2019_7A40_EA5412513C5A'}
	(* Equalize the histogram of a grayscale or color image, which normalizes the brightness and improves the contrast. (expert function) 
	The channel index that should be equalized has to be specified (-1 expects a RGB image, converts it to YCbCr, equalizes the Y channel and converts the image back to RGB).  *)
	FUNCTION F_VN_HistogramEqualizationExp : HRESULT
	VAR_INPUT
		ipSrcImage	:	ITcVnImage;	(* Source image (USINT) *)
		ipDestImage	:	REFERENCE TO ITcVnImage;	(* Destination image (An appropriate destination image will be created if required.) *)
		nChannelIdx	:	INT;	(* Index of the image channel that should be equalized (-1 expects a RGB image, converts it to YCbCr, equalizes the Y channel and converts the image back to RGB) *)
		hrPrev	:	HRESULT;	(* HRESULT indicating the result of previous operations (If SUCCEEDED(hrPrev) equals false, no operation is executed.) *)
	END_VAR

END_FUNCTION

// Functions/Image Color and Contrast Processing/F_VN_InvertImageColor

	{attribute 'TcIecLibraryType'}
	{attribute 'external_name' := 'F_VN_InvertImageColor_GUID_6A9DE08A_3024_20D5_5961_946D9F73E371'}
	(* Invert the color of an image.
          For signed integer or negative floating point values, only the signs will be switched.
          If the image contains only positive floating point values, each pixel value is subtracted from the maximum available pixel value (or 1.0, whatever is higher). *)
	FUNCTION F_VN_InvertImageColor : HRESULT
	VAR_INPUT
		ipSrcImage	:	ITcVnImage;	(* Source image *)
		ipDestImage	:	REFERENCE TO ITcVnImage;	(* Destination image (An appropriate image will be created if required.) *)
		hrPrev	:	HRESULT;	(* HRESULT indicating the result of previous operations (If SUCCEEDED(hrPrev) equals false, no operation is executed.) *)
	END_VAR

END_FUNCTION

// Functions/Image Color and Contrast Processing/F_VN_InvertImageColorExp

	{attribute 'TcIecLibraryType'}
	{attribute 'external_name' := 'F_VN_InvertImageColorExp_GUID_85EBF390_511C_207F_6A2E_C8823AF722BD'}
	(* Invert the color of an image. (expert function)
          For signed integer or negative floating point values, only the signs will be switched.
          If the image contains only positive floating point values, each pixel value is subtracted from the maximum available pixel value (or 1.0, whatever is higher). *)
	FUNCTION F_VN_InvertImageColorExp : HRESULT
	VAR_INPUT
		ipSrcImage	:	ITcVnImage;	(* Source image *)
		ipDestImage	:	REFERENCE TO ITcVnImage;	(* Destination image (An appropriate image will be created if required.) *)
		fMaxValue	:	LREAL;	(* Maximum pixel value (e.g. if a 16 bit image contains 12 bit values). -1 means the default values are used. *)
		hrPrev	:	HRESULT;	(* HRESULT indicating the result of previous operations (If SUCCEEDED(hrPrev) equals false, no operation is executed.) *)
	END_VAR

END_FUNCTION

// Functions/Image Color and Contrast Processing/F_VN_NormalizeImage

	{attribute 'TcIecLibraryType'}
	{attribute 'external_name' := 'F_VN_NormalizeImage_GUID_5CE899FF_D18C_217F_632A_AAB18A76EAE9'}
	(* Normalize an image regarding its value range (e.g. stretch pixel values [50..150] to full range [0..255]). *)
	FUNCTION F_VN_NormalizeImage : HRESULT
	VAR_INPUT
		ipSrcImage	:	ITcVnImage;	(* Source image *)
		ipDestImage	:	REFERENCE TO ITcVnImage;	(* Destination image (An appropriate destination image will be created if required.) *)
		hrPrev	:	HRESULT;	(* HRESULT indicating the result of previous operations (If SUCCEEDED(hrPrev) equals false, no operation is executed.) *)
	END_VAR

END_FUNCTION

// Functions/Image Color and Contrast Processing/F_VN_NormalizeImageExp

	{attribute 'TcIecLibraryType'}
	{attribute 'external_name' := 'F_VN_NormalizeImageExp_GUID_A404DE13_94C0_24F5_463B_0CBCEE4D30A5'}
	(* Normalize an image regarding its value range (e.g. stretch pixel values [50..150] to full range [0..255]) or scale the values regarding a specific normalization (e.g. L2-norm). (expert function) *)
	FUNCTION F_VN_NormalizeImageExp : HRESULT
	VAR_INPUT
		ipSrcImage	:	ITcVnImage;	(* Source image *)
		ipDestImage	:	REFERENCE TO ITcVnImage;	(* Destination image (An appropriate destination image will be created if required.) *)
		fAlpha	:	LREAL;	(* Lower range boundary (in case of normalizing the value range) or value to normalize to (||ipDestImage|| = fAlpha) *)
		fBeta	:	LREAL;	(* Upper range boundary (in case of normalizing the value range) *)
		eNormType	:	ETcVnNormalizationType;	(* Normalization type (only INF, L1, L2 or MINMAX) *)
		eDestType	:	ETcVnElementType;	(* Destination image depth (usually SAME_AS_SOURCE) *)
		ipMask	:	ITcVnImage;	(* Mask to restrict the normalization to specific pixel positions (set 0 to normalize the whole image) *)
		hrPrev	:	HRESULT;	(* HRESULT indicating the result of previous operations (If SUCCEEDED(hrPrev) equals false, no operation is executed.) *)
	END_VAR

END_FUNCTION

// Functions/Image Color and Contrast Processing/F_VN_NormalizeImageForDisplay

	{attribute 'TcIecLibraryType'}
	{attribute 'external_name' := 'F_VN_NormalizeImageForDisplay_GUID_07187A7C_1E4E_2D22_6499_C2CF63C81977'}
	(* Normalize an image for display, i.e. scale it to the full value range of the underlying data type (-1 to 1 for floating point). *)
	FUNCTION F_VN_NormalizeImageForDisplay : HRESULT
	VAR_INPUT
		ipSrcImage	:	ITcVnImage;	(* Source image *)
		ipDestImage	:	REFERENCE TO ITcVnImage;	(* Destination image (An appropriate destination image will be created if required.) *)
		eSignedNormalization	:	ETcVnSignedNormalization;	(* Option for normalizing signed values *)
		hrPrev	:	HRESULT;	(* HRESULT indicating the result of previous operations (If SUCCEEDED(hrPrev) equals false, no operation is executed.) *)
	END_VAR

END_FUNCTION

// Functions/Image Color and Contrast Processing/F_VN_ReferenceColorSimilarity_ITcVnColorModel

	{attribute 'TcIecLibraryType'}
	{attribute 'external_name' := 'F_VN_ReferenceColorSimilarity_ITcVnColorModel_GUID_773EAF27_B6E6_2465_5C4F_FC1E2678EDFA'}
	(* Computes the similarity to a reference color model for each pixel in the source image. *)
	FUNCTION F_VN_ReferenceColorSimilarity_ITcVnColorModel : HRESULT
	VAR_INPUT
		ipSrcImage	:	ITcVnImage;	(* RGB source image (USINT, 3 channels) *)
		ipDestImage	:	REFERENCE TO ITcVnImage;	(* Returns the similarity to ipColorModel for each pixel in ipSrcImage (USINT, 1 channel. An appropriate destination image will be created if required.) *)
		ipColorModel	:	ITcVnColorModel;	(* Color model *)
		hrPrev	:	HRESULT;	(* HRESULT indicating the result of previous operations (If SUCCEEDED(hrPrev) equals false, no operation is executed.) *)
	END_VAR

END_FUNCTION

// Interfaces/Machine Learning/ITcVnColorModel

	(* Interface to train and classify an image color. *)
	{attribute 'c++_compatible'}
	{attribute 'vtable_order' := 'TrainImageColor;ClassifyImageColor'}
	INTERFACE ITcVnColorModel EXTENDS ITcVnMlModel


(* Train the color of the provided image. *)
	{attribute 'c++_compatible'}
	{attribute 'minimal_input_size' := '4'}
	{attribute 'pack_mode' := '4'}
	METHOD TrainImageColor : HRESULT
	VAR_INPUT
		ipSrcImage : ITcVnImage;
		nDifferentColors : UDINT;
		ipMask : ITcVnImage;
		nSkipPixels : UDINT;
	END_VAR
END_METHOD


(* Compute the similarity of each image pixel to the trained reference color. *)
	{attribute 'c++_compatible'}
	{attribute 'minimal_input_size' := '4'}
	{attribute 'pack_mode' := '4'}
	METHOD ClassifyImageColor : HRESULT
	VAR_INPUT
		ipSrcImage : ITcVnImage;
		pipDestImage : POINTER TO ITcVnImage;
		fVariance : REAL;
		fLuminanceWeight : REAL;
	END_VAR
END_METHOD

END_INTERFACE

// Functions/Image Color and Contrast Processing/F_VN_ReferenceColorSimilarityExp_ITcVnColorModel

	{attribute 'TcIecLibraryType'}
	{attribute 'external_name' := 'F_VN_ReferenceColorSimilarityExp_ITcVnColorModel_GUID_73229F9C_3F17_25D2_76F6_22BB9B62AC8E'}
	(* Computes the similarity to a reference color model for each pixel in the source image. (expert function) *)
	FUNCTION F_VN_ReferenceColorSimilarityExp_ITcVnColorModel : HRESULT
	VAR_INPUT
		ipSrcImage	:	ITcVnImage;	(* RGB source image (USINT, 3 channels) *)
		ipDestImage	:	REFERENCE TO ITcVnImage;	(* Returns the similarity to ipColorModel for each pixel in ipSrcImage (USINT, 1 channel. An appropriate destination image will be created if required.) *)
		ipColorModel	:	ITcVnColorModel;	(* Color model *)
		fVariance	:	REAL;	(* Allowed color variance (0.1 - 0.3 might be a good start to try) *)
		fLuminanceWeight	:	REAL;	(* Weight the impact of the luminance ([0..1], e.g. set to 0 to be more resistant to unequal illumination, but might be required to differentiate between some colors. Ignored if ipColorModel is of type RGB.) *)
		hrPrev	:	HRESULT;	(* HRESULT indicating the result of previous operations (If SUCCEEDED(hrPrev) equals false, no operation is executed.) *)
	END_VAR

END_FUNCTION

// Functions/Image Color and Contrast Processing/F_VN_ReferenceColorSimilarity_ITcVnMlModel

	{attribute 'TcIecLibraryType'}
	{attribute 'external_name' := 'F_VN_ReferenceColorSimilarity_ITcVnMlModel_GUID_2753D489_F47A_2B57_6B29_1A2D331DDEEE'}
	(* Computes the similarity to a reference color model for each pixel in the source image. *)
	FUNCTION F_VN_ReferenceColorSimilarity_ITcVnMlModel : HRESULT
	VAR_INPUT
		ipSrcImage	:	ITcVnImage;	(* RGB source image (USINT, 3 channels) *)
		ipDestImage	:	REFERENCE TO ITcVnImage;	(* Returns the similarity to ipColorModel for each pixel in ipSrcImage (USINT, 1 channel. An appropriate destination image will be created if required.) *)
		ipColorModel	:	ITcVnMlModel;	(* Color model *)
		hrPrev	:	HRESULT;	(* HRESULT indicating the result of previous operations (If SUCCEEDED(hrPrev) equals false, no operation is executed.) *)
	END_VAR

END_FUNCTION

// Functions/Image Color and Contrast Processing/F_VN_ReferenceColorSimilarityExp_ITcVnMlModel

	{attribute 'TcIecLibraryType'}
	{attribute 'external_name' := 'F_VN_ReferenceColorSimilarityExp_ITcVnMlModel_GUID_058FAC2B_F274_2EC2_5B40_C884C3F350AB'}
	(* Computes the similarity to a reference color model for each pixel in the source image. (expert function) *)
	FUNCTION F_VN_ReferenceColorSimilarityExp_ITcVnMlModel : HRESULT
	VAR_INPUT
		ipSrcImage	:	ITcVnImage;	(* RGB source image (USINT, 3 channels) *)
		ipDestImage	:	REFERENCE TO ITcVnImage;	(* Returns the similarity to ipColorModel for each pixel in ipSrcImage (USINT, 1 channel. An appropriate destination image will be created if required.) *)
		ipColorModel	:	ITcVnMlModel;	(* Color model *)
		fVariance	:	REAL;	(* Allowed color variance (0.1 - 0.3 might be a good start to try) *)
		fLuminanceWeight	:	REAL;	(* Weight the impact of the luminance ([0..1], e.g. set to 0 to be more resistant to unequal illumination, but might be required to differentiate between some colors. Ignored if ipColorModel is of type RGB.) *)
		hrPrev	:	HRESULT;	(* HRESULT indicating the result of previous operations (If SUCCEEDED(hrPrev) equals false, no operation is executed.) *)
	END_VAR

END_FUNCTION

// Functions/Image Color and Contrast Processing/F_VN_ReferenceColorSimilarity_TcVnVector3_LREAL

	{attribute 'TcIecLibraryType'}
	{attribute 'external_name' := 'F_VN_ReferenceColorSimilarity_TcVnVector3_LREAL_GUID_A7DE5E54_87EA_2D91_638A_0808EFE078D5'}
	(* Computes the similarity to a reference color for each pixel in the source image. *)
	FUNCTION F_VN_ReferenceColorSimilarity_TcVnVector3_LREAL : HRESULT
	VAR_INPUT
		ipSrcImage	:	ITcVnImage;	(* RGB source image (USINT, 3 channels) *)
		ipDestImage	:	REFERENCE TO ITcVnImage;	(* Returns the similarity to aRefColor for each pixel in ipSrcImage (USINT, 1 channel. An appropriate destination image will be created if required.) *)
	END_VAR
	VAR_IN_OUT
		aRefColor	:	TcVnVector3_LREAL;	(* Reference color (RGB, [0..255]) *)
	END_VAR
	VAR_INPUT
		hrPrev	:	HRESULT;	(* HRESULT indicating the result of previous operations (If SUCCEEDED(hrPrev) equals false, no operation is executed.) *)
	END_VAR

END_FUNCTION

// Functions/Image Color and Contrast Processing/F_VN_ReferenceColorSimilarityExp_TcVnVector3_LREAL

	{attribute 'TcIecLibraryType'}
	{attribute 'external_name' := 'F_VN_ReferenceColorSimilarityExp_TcVnVector3_LREAL_GUID_8E557551_A40C_2744_5752_5B1B0681E0C1'}
	(* Computes the similarity to a reference color for each pixel in the source image. (expert function) *)
	FUNCTION F_VN_ReferenceColorSimilarityExp_TcVnVector3_LREAL : HRESULT
	VAR_INPUT
		ipSrcImage	:	ITcVnImage;	(* RGB source image (USINT, 3 channels) *)
		ipDestImage	:	REFERENCE TO ITcVnImage;	(* Returns the similarity to aRefColor for each pixel in ipSrcImage (USINT, 1 channel. An appropriate destination image will be created if required.) *)
	END_VAR
	VAR_IN_OUT
		aRefColor	:	TcVnVector3_LREAL;	(* Reference color (RGB, [0..255]) *)
	END_VAR
	VAR_INPUT
		fVariance	:	REAL;	(* Allowed color variance (0.1 - 0.3 might be a good start to try) *)
		fLuminanceWeight	:	REAL;	(* Weight the impact of the luminance ([0..1], e.g. set to 0 to be more resistant to unequal illumination, but might be required to differentiate between some colors) *)
		hrPrev	:	HRESULT;	(* HRESULT indicating the result of previous operations (If SUCCEEDED(hrPrev) equals false, no operation is executed.) *)
	END_VAR

END_FUNCTION

// Functions/Image Color and Contrast Processing/F_VN_TrainImageColor

	{attribute 'TcIecLibraryType'}
	{attribute 'external_name' := 'F_VN_TrainImageColor_GUID_5FA703BF_81EA_2D0C_57DC_D3E884560665'}
	(* Create a new color model, describing the image color. *)
	FUNCTION F_VN_TrainImageColor : HRESULT
	VAR_INPUT
		ipSrcImage	:	ITcVnImage;	(* Source image (3 channels (RGB) of type USINT) *)
		ipColorModel	:	REFERENCE TO ITcVnColorModel;	(* Returns the color model *)
		nDifferentColors	:	UDINT;	(* Number of different colors to distinguish *)
		hrPrev	:	HRESULT;	(* HRESULT indicating the result of previous operations (If SUCCEEDED(hrPrev) equals false, no operation is executed.) *)
	END_VAR

END_FUNCTION

// Functions/Image Color and Contrast Processing/F_VN_TrainImageColorExp

	{attribute 'TcIecLibraryType'}
	{attribute 'external_name' := 'F_VN_TrainImageColorExp_GUID_3C728016_1A49_2A7E_70C2_8FAE5DF32F9C'}
	(* Create a new color model, describing the image color. (expert function) *)
	FUNCTION F_VN_TrainImageColorExp : HRESULT
	VAR_INPUT
		ipSrcImage	:	ITcVnImage;	(* Source image (3 channels (RGB) of type USINT) *)
		ipColorModel	:	REFERENCE TO ITcVnColorModel;	(* Returns the color model *)
		nDifferentColors	:	UDINT;	(* Number of different colors to distinguish *)
		eMethod	:	ETcVnColorTrainingMethod;	(* Color training method *)
		ipMask	:	ITcVnImage;	(* Optional image mask (1 channel of type USINT, set to 0 if not required) *)
		nSkipPixels	:	UDINT;	(* Number of pixels to skip between each evaluated color sample (to achieve a better performance). 0 takes every pixel into account and tends to be more accurate. *)
		hrPrev	:	HRESULT;	(* HRESULT indicating the result of previous operations (If SUCCEEDED(hrPrev) equals false, no operation is executed.) *)
	END_VAR

END_FUNCTION

// Functions/Image Color and Contrast Processing/F_VN_TrainImageColorExp2

	{attribute 'TcIecLibraryType'}
	{attribute 'external_name' := 'F_VN_TrainImageColorExp2_GUID_5943C5EF_12AF_22DC_62B5_F2E4E5724ACA'}
	(* Create a new color model, describing the image color. (expert function) *)
	FUNCTION F_VN_TrainImageColorExp2 : HRESULT
	VAR_INPUT
		ipSrcImage	:	ITcVnImage;	(* Source image (3 channels (RGB) of type USINT) *)
		ipColorModel	:	REFERENCE TO ITcVnColorModel;	(* Returns the color model *)
		nDifferentColors	:	UDINT;	(* Maximum number of different colors to distinguish (if LBG is used as a clustering algorithm, the result might have less different colors, depending on nMaxClusterRadius) *)
		eMethod	:	ETcVnColorTrainingMethod;	(* Color training method *)
		ipMask	:	ITcVnImage;	(* Optional image mask (1 channel of type USINT, set to 0 if not required) *)
		nSkipPixels	:	UDINT;	(* Number of pixels to skip between each evaluated color sample (to achieve a better performance). 0 takes every pixel into account and tends to be more accurate. *)
		eClusteringAlgorithm	:	ETcVnClusteringAlgorithm;	(* Clustering algorithm *)
		nMaxClusterRadius	:	DINT;	(* Only used for the LBG clustering algorithm. Maximum allowed radius (> 0) of a single cluster, i.e. clusters with a higher radius will be split into smaller ones, until a global number of nDifferentColors is reached. *)
		bSingleSplitSteps	:	BOOL;	(* Only used for the LBG clustering algorithm. If true, the global optimization is always run after a single cluster has been split. If false, several clusters are split within the same step before applying the global optimization. Applying the global optimization less often is faster, but can lead to less optimal results, especially having 2 nearby clusters that could be represented by 1) *)
		hrPrev	:	HRESULT;	(* HRESULT indicating the result of previous operations (If SUCCEEDED(hrPrev) equals false, no operation is executed.) *)
	END_VAR

END_FUNCTION

// Functions/Image Color and Contrast Processing/F_VN_TrainImageColor_ITcVnMlModel

	{attribute 'TcIecLibraryType'}
	{attribute 'external_name' := 'F_VN_TrainImageColor_ITcVnMlModel_GUID_14A403BF_02E9_2A86_65F6_90D5E015B862'}
	(* Create a new color model, describing the image color. *)
	FUNCTION F_VN_TrainImageColor_ITcVnMlModel : HRESULT
	VAR_INPUT
		ipSrcImage	:	ITcVnImage;	(* Source image (3 channels (RGB) of type USINT) *)
		ipColorModel	:	REFERENCE TO ITcVnMlModel;	(* Returns the color model *)
		nDifferentColors	:	UDINT;	(* Number of different colors to distinguish *)
		hrPrev	:	HRESULT;	(* HRESULT indicating the result of previous operations (If SUCCEEDED(hrPrev) equals false, no operation is executed.) *)
	END_VAR

END_FUNCTION

// Functions/Image Color and Contrast Processing/F_VN_TrainImageColorExp_ITcVnMlModel

	{attribute 'TcIecLibraryType'}
	{attribute 'external_name' := 'F_VN_TrainImageColorExp_ITcVnMlModel_GUID_B74A77B1_4DA0_2812_5AE5_3A16426A639C'}
	(* Create a new color model, describing the image color. (expert function) *)
	FUNCTION F_VN_TrainImageColorExp_ITcVnMlModel : HRESULT
	VAR_INPUT
		ipSrcImage	:	ITcVnImage;	(* Source image (3 channels (RGB) of type USINT) *)
		ipColorModel	:	REFERENCE TO ITcVnMlModel;	(* Returns the color model *)
		nDifferentColors	:	UDINT;	(* Number of different colors to distinguish *)
		eMethod	:	ETcVnColorTrainingMethod;	(* Color training method *)
		ipMask	:	ITcVnImage;	(* Optional image mask (1 channel of type USINT, set to 0 if not required) *)
		nSkipPixels	:	UDINT;	(* Number of pixels to skip between each evaluated color sample (to achieve a better performance). 0 takes every pixel into account and tends to be more accurate. *)
		hrPrev	:	HRESULT;	(* HRESULT indicating the result of previous operations (If SUCCEEDED(hrPrev) equals false, no operation is executed.) *)
	END_VAR

END_FUNCTION

// Functions/Image Color and Contrast Processing/F_VN_TrainImageColorExp2_ITcVnMlModel

	{attribute 'TcIecLibraryType'}
	{attribute 'external_name' := 'F_VN_TrainImageColorExp2_ITcVnMlModel_GUID_0F70CC6A_E154_20C7_6938_0B7E87ECC22B'}
	(* Create a new color model, describing the image color. (expert function) *)
	FUNCTION F_VN_TrainImageColorExp2_ITcVnMlModel : HRESULT
	VAR_INPUT
		ipSrcImage	:	ITcVnImage;	(* Source image (3 channels (RGB) of type USINT) *)
		ipColorModel	:	REFERENCE TO ITcVnMlModel;	(* Returns the color model *)
		nDifferentColors	:	UDINT;	(* Maximum number of different colors to distinguish (if LBG is used as a clustering algorithm, the result might have less different colors, depending on nMaxClusterRadius) *)
		eMethod	:	ETcVnColorTrainingMethod;	(* Color training method *)
		ipMask	:	ITcVnImage;	(* Optional image mask (1 channel of type USINT, set to 0 if not required) *)
		nSkipPixels	:	UDINT;	(* Number of pixels to skip between each evaluated color sample (to achieve a better performance). 0 takes every pixel into account and tends to be more accurate. *)
		eClusteringAlgorithm	:	ETcVnClusteringAlgorithm;	(* Clustering algorithm *)
		nMaxClusterRadius	:	DINT;	(* Only used for the LBG clustering algorithm. Maximum allowed radius (> 0) of a single cluster, i.e. clusters with a higher radius will be split into smaller ones, until a global number of nDifferentColors is reached. *)
		bSingleSplitSteps	:	BOOL;	(* Only used for the LBG clustering algorithm. If true, the global optimization is always run after a single cluster has been split. If false, several clusters are split within the same step before applying the global optimization. Applying the global optimization less often is faster, but can lead to less optimal results, especially having 2 nearby clusters that could be represented by 1) *)
		hrPrev	:	HRESULT;	(* HRESULT indicating the result of previous operations (If SUCCEEDED(hrPrev) equals false, no operation is executed.) *)
	END_VAR

END_FUNCTION

// Functions/Image Color and Contrast Processing/F_VN_WhiteBalance

	{attribute 'TcIecLibraryType'}
	{attribute 'external_name' := 'F_VN_WhiteBalance_GUID_C72124E6_44C4_22B6_45BC_08CB003F8D94'}
	(* Calculates the white balance ratios for a RGB image. Uses the green channel as a reference and computes the relative ratios for the red and blue channels. Requires a non-reflecting, not overexposed white colored object (e.g. a sheet of paper) in at least 100 pixels of the image to provide reasonable results. The resulting ratios can then be set on the camera (multiply with existing ratios), or applied in the PLC via MultiplyImageWithVector. *)
	FUNCTION F_VN_WhiteBalance : HRESULT
	VAR_INPUT
		ipSrcImage	:	ITcVnImage;	(* Source image (3 channels (RGB), USINT or UINT) *)
		ipDestImage	:	REFERENCE TO ITcVnImage;	(* Destination image with white balance applied (optional, set to 0 if not required. An appropriate image will be created if required.) *)
		fRatioRed	:	REFERENCE TO REAL;	(* Returns the ratio for the red channel *)
		fRatioBlue	:	REFERENCE TO REAL;	(* Returns the ratio for the blue channel *)
		nMaxValue	:	UDINT;	(* Specify the maximum pixel value that would be achieved by overexposure (usually 255 for 8 bit or 4095 for 12 bit data) *)
		hrPrev	:	HRESULT;	(* HRESULT indicating the result of previous operations (If SUCCEEDED(hrPrev) equals false, no operation is executed.) *)
	END_VAR

END_FUNCTION

// Functions/Contour Analysis/F_VN_ApproximatePolygon

	{attribute 'TcIecLibraryType'}
	{attribute 'external_name' := 'F_VN_ApproximatePolygon_GUID_FB544BB9_796A_2F50_6D99_3E70FEF2DD64'}
	(* Approximate a contour to a simplified polygon (using the Douglas-Peucker algorithm). *)
	FUNCTION F_VN_ApproximatePolygon : HRESULT
	VAR_INPUT
		ipSrcContour	:	ITcVnContainer;	(* Single contour (ContainerType_Vector_TcVnPoint2_DINT or ContainerType_Vector_TcVnPoint2_REAL; The elements of this container are the points of the contour.) *)
		ipDestContour	:	REFERENCE TO ITcVnContainer;	(* Returns a container which is filled with the approximated polygon points (same type ID as ipSrcContour; Non-zero interface pointers are reused.) *)
		fMaxDist	:	LREAL;	(* Maximum distance between the original contour and its approximation *)
		bClosed	:	BOOL;	(* Specify, if the contour is closed (first and last points connected) or not *)
		hrPrev	:	HRESULT;	(* HRESULT indicating the result of previous operations (If SUCCEEDED(hrPrev) equals false, no operation is executed.) *)
	END_VAR

END_FUNCTION

// Functions/Contour Analysis/F_VN_CheckIfPointIsInsideContour

	{attribute 'TcIecLibraryType'}
	{attribute 'external_name' := 'F_VN_CheckIfPointIsInsideContour_GUID_3E514BE2_7E1F_213B_7184_D29B7EA6D7D6'}
	(* Checks if a point is inside a contour (and optionally return the distance to it). *)
	FUNCTION F_VN_CheckIfPointIsInsideContour : HRESULT
	VAR_INPUT
		ipContour	:	ITcVnContainer;	(* Single contour (ContainerType_Vector_TcVnPoint2_DINT or ContainerType_Vector_TcVnPoint2_REAL) *)
	END_VAR
	VAR_IN_OUT
		aPoint	:	TcVnPoint2_REAL;	(* Point position to check *)
		fDist	:	LREAL;	(* Returns the result (> 0: the point is inside the contour; 0: the point is on the contour; < 0: the point is outside the contour) *)
	END_VAR
	VAR_INPUT
		bMeasureDistance	:	BOOL;	(* If true, fDist returns the distance to the nearest contour edge. Otherwise, fDist only returns -1, 0 or +1 (recommended to set to false if the distance is not required, as this is faster). *)
		hrPrev	:	HRESULT;	(* HRESULT indicating the result of previous operations (If SUCCEEDED(hrPrev) equals false, no operation is executed.) *)
	END_VAR

END_FUNCTION

// Functions/Contour Analysis/F_VN_ContourArea

	{attribute 'TcIecLibraryType'}
	{attribute 'external_name' := 'F_VN_ContourArea_GUID_EF9B112B_FB92_2835_5B41_8807AFE46848'}
	(* Estimate the contour area using Green's formula. *)
	FUNCTION F_VN_ContourArea : HRESULT
	VAR_INPUT
		ipContour	:	ITcVnContainer;	(* Single contour (ContainerType_Vector_TcVnPoint2_DINT or ContainerType_Vector_TcVnPoint2_REAL; The elements of this container are the points of the contour.) *)
	END_VAR
	VAR_IN_OUT
		fArea	:	LREAL;	(* Returns the estimated contour area (The actual contour area may differ depending on the shape of the contour.) *)
	END_VAR
	VAR_INPUT
		hrPrev	:	HRESULT;	(* HRESULT indicating the result of previous operations (If SUCCEEDED(hrPrev) equals false, no operation is executed.) *)
	END_VAR

END_FUNCTION

// Functions/Contour Analysis/F_VN_ContourCenterOfMass

	{attribute 'TcIecLibraryType'}
	{attribute 'external_name' := 'F_VN_ContourCenterOfMass_GUID_53FF4B7A_5FC7_2CCA_4C08_7EE432242F75'}
	(* Computes the center of mass of a contour. *)
	FUNCTION F_VN_ContourCenterOfMass : HRESULT
	VAR_INPUT
		ipContour	:	ITcVnContainer;	(* Single contour (ContainerType_Vector_TcVnPoint2_DINT or ContainerType_Vector_TcVnPoint2_REAL; The elements of this container are the points of the contour.) *)
	END_VAR
	VAR_IN_OUT
		aCenterOfMass	:	TcVnPoint2_LREAL;	(* Returns the center of mass of the contour *)
	END_VAR
	VAR_INPUT
		hrPrev	:	HRESULT;	(* HRESULT indicating the result of previous operations (If SUCCEEDED(hrPrev) equals false, no operation is executed.) *)
	END_VAR

END_FUNCTION

// Functions/Contour Analysis/F_VN_ContourCircularity

	{attribute 'TcIecLibraryType'}
	{attribute 'external_name' := 'F_VN_ContourCircularity_GUID_A914FD7D_5A40_2400_42D0_7DA47E4F4D53'}
	(* Computes the circularity of a contour (1.0: ideal circle, 0.0: straight line). *)
	FUNCTION F_VN_ContourCircularity : HRESULT
	VAR_INPUT
		ipContour	:	ITcVnContainer;	(* Single contour (ContainerType_Vector_TcVnPoint2_DINT or ContainerType_Vector_TcVnPoint2_REAL; The elements of this container are the points of the contour.) *)
	END_VAR
	VAR_IN_OUT
		fCircularity	:	LREAL;	(* Returns the circularity of the contour [0..1] *)
	END_VAR
	VAR_INPUT
		hrPrev	:	HRESULT;	(* HRESULT indicating the result of previous operations (If SUCCEEDED(hrPrev) equals false, no operation is executed.) *)
	END_VAR

END_FUNCTION

// Functions/Contour Analysis/F_VN_ContourCircularityExp

	{attribute 'TcIecLibraryType'}
	{attribute 'external_name' := 'F_VN_ContourCircularityExp_GUID_D9CDD8B0_F351_2C6F_6BB7_A742C5ADB59D'}
	(* Computes the circularity of a contour (1.0: ideal circle, 0.0: straight line). (expert function) *)
	FUNCTION F_VN_ContourCircularityExp : HRESULT
	VAR_INPUT
		ipContour	:	ITcVnContainer;	(* Single contour (ContainerType_Vector_TcVnPoint2_DINT or ContainerType_Vector_TcVnPoint2_REAL; The elements of this container are the points of the contour.) *)
	END_VAR
	VAR_IN_OUT
		fCircularity	:	LREAL;	(* Returns the circularity of the contour [0..1] *)
	END_VAR
	VAR_INPUT
		eMethod	:	ETcVnCircularityCalculationMethod;	(* Method used for computing the circularity *)
		hrPrev	:	HRESULT;	(* HRESULT indicating the result of previous operations (If SUCCEEDED(hrPrev) equals false, no operation is executed.) *)
	END_VAR

END_FUNCTION

// Functions/Contour Analysis/F_VN_ContourConvexity

	{attribute 'TcIecLibraryType'}
	{attribute 'external_name' := 'F_VN_ContourConvexity_GUID_477A673C_7DC9_2383_6476_7BD35E49CD18'}
	(* Computes the convexity of a contour as the ratio between the contour's area and the area of the convex hull (1.0: convex shapes (i.e. rectangle, circle, ..., etc.), 0.0: zero area (i.e. a line or an empty contour)). *)
	FUNCTION F_VN_ContourConvexity : HRESULT
	VAR_INPUT
		ipContour	:	ITcVnContainer;	(* Single contour (ContainerType_Vector_TcVnPoint2_DINT or ContainerType_Vector_TcVnPoint2_REAL; The elements of this container are the points of the contour.) *)
	END_VAR
	VAR_IN_OUT
		fConvexity	:	LREAL;	(* Returns the convexity of the contour [0..1] *)
	END_VAR
	VAR_INPUT
		hrPrev	:	HRESULT;	(* HRESULT indicating the result of previous operations (If SUCCEEDED(hrPrev) equals false, no operation is executed.) *)
	END_VAR

END_FUNCTION

// Functions/Contour Analysis/F_VN_ContourEccentricity

	{attribute 'TcIecLibraryType'}
	{attribute 'external_name' := 'F_VN_ContourEccentricity_GUID_C8A66092_AFCE_2D41_6EFC_D440ACB58899'}
	(* Computes the eccentricity of a contour (0.0: circular, 1.0: linear). *)
	FUNCTION F_VN_ContourEccentricity : HRESULT
	VAR_INPUT
		ipContour	:	ITcVnContainer;	(* Single contour (ContainerType_Vector_TcVnPoint2_DINT or ContainerType_Vector_TcVnPoint2_REAL; The elements of this container are the points of the contour.) *)
	END_VAR
	VAR_IN_OUT
		fEccentricity	:	LREAL;	(* Returns the eccentricity of the contour [0..1] *)
	END_VAR
	VAR_INPUT
		hrPrev	:	HRESULT;	(* HRESULT indicating the result of previous operations (If SUCCEEDED(hrPrev) equals false, no operation is executed.) *)
	END_VAR

END_FUNCTION

// Functions/Contour Analysis/F_VN_ContourElongation

	{attribute 'TcIecLibraryType'}
	{attribute 'external_name' := 'F_VN_ContourElongation_GUID_65A1F331_73BE_2BA2_68E7_E3CB51703C65'}
	(* Computes the elongation factor of a contour. *)
	FUNCTION F_VN_ContourElongation : HRESULT
	VAR_INPUT
		ipContour	:	ITcVnContainer;	(* Single contour (ContainerType_Vector_TcVnPoint2_DINT or ContainerType_Vector_TcVnPoint2_REAL; The elements of this container are the points of the contour.) *)
	END_VAR
	VAR_IN_OUT
		fElongation	:	LREAL;	(* Returns the elongation of the contour *)
	END_VAR
	VAR_INPUT
		hrPrev	:	HRESULT;	(* HRESULT indicating the result of previous operations (If SUCCEEDED(hrPrev) equals false, no operation is executed.) *)
	END_VAR

END_FUNCTION

// Functions/Contour Analysis/F_VN_ContourExtremePoint

	{attribute 'TcIecLibraryType'}
	{attribute 'external_name' := 'F_VN_ContourExtremePoint_GUID_B802725E_49B6_2206_63CD_CF23A01B9AB2'}
	(* Finds the contour extreme point. *)
	FUNCTION F_VN_ContourExtremePoint : HRESULT
	VAR_INPUT
		ipContour	:	ITcVnContainer;	(* Source container with 2D points (TcVnPoint2_DINT or TcVnPoint2_REAL or TcVnPoint2_LREAL) *)
		eDirection	:	ETcVnExtremePointDirection;	(* Selects the search direction for the extreme point *)
	END_VAR
	VAR_IN_OUT
		aExtremePoint	:	TcVnPoint2_LREAL;	(* Returns the extreme point of the contour, according to eDirection *)
	END_VAR
	VAR_INPUT
		hrPrev	:	HRESULT;	(* HRESULT indicating the result of previous operations (If SUCCEEDED(hrPrev) equals false, no operation is executed.) *)
	END_VAR

END_FUNCTION

// Functions/Contour Analysis/F_VN_ContourInertiaRatio

	{attribute 'TcIecLibraryType'}
	{attribute 'external_name' := 'F_VN_ContourInertiaRatio_GUID_A0B90893_4522_2D9E_7968_93574BE8615A'}
	(* Computes the inertia ratio of a contour which reflects how a contour/shape is elongated (i.e. circle: 1.0, line: 0.0). *)
	FUNCTION F_VN_ContourInertiaRatio : HRESULT
	VAR_INPUT
		ipContour	:	ITcVnContainer;	(* Single contour (ContainerType_Vector_TcVnPoint2_DINT or ContainerType_Vector_TcVnPoint2_REAL; The elements of this container are the points of the contour.) *)
	END_VAR
	VAR_IN_OUT
		fInertiaRatio	:	LREAL;	(* Returns the inertia raio of the contour [0..1] *)
	END_VAR
	VAR_INPUT
		hrPrev	:	HRESULT;	(* HRESULT indicating the result of previous operations (If SUCCEEDED(hrPrev) equals false, no operation is executed.) *)
	END_VAR

END_FUNCTION

// Functions/Contour Analysis/F_VN_ContourMoments

	{attribute 'TcIecLibraryType'}
	{attribute 'external_name' := 'F_VN_ContourMoments_GUID_CDBD8489_7323_25E5_6FE9_D32063BF7695'}
	(* Computes the spatial moments, the central moments, and the central normalized moments of a contour up to the third order. *)
	FUNCTION F_VN_ContourMoments : HRESULT
	VAR_INPUT
		ipContour	:	ITcVnContainer;	(* Single contour (ContainerType_Vector_TcVnPoint2_DINT or ContainerType_Vector_TcVnPoint2_REAL; The elements of this container are the points of the contour.) *)
	END_VAR
	VAR_IN_OUT
		stMoments	:	TcVnMoments;	(* Returns a struct containing the moments *)
	END_VAR
	VAR_INPUT
		hrPrev	:	HRESULT;	(* HRESULT indicating the result of previous operations (If SUCCEEDED(hrPrev) equals false, no operation is executed.) *)
	END_VAR

END_FUNCTION

// Functions/Contour Analysis/F_VN_ContourOrientation

	{attribute 'TcIecLibraryType'}
	{attribute 'external_name' := 'F_VN_ContourOrientation_GUID_B9BAE3E9_19EE_2785_58C6_96C4C45F52E5'}
	(* Calculate the orientation of a contour or a set of points. *)
	FUNCTION F_VN_ContourOrientation : HRESULT
	VAR_INPUT
		ipContour	:	ITcVnContainer;	(* Source point set (ContainerType_Vector_TcVnPoint2_DINT, ContainerType_Vector_TcVnPoint2_REAL, or ContainerType_Vector_TcVnPoint2_LREAL. The elements of this container are the individual points.) *)
	END_VAR
	VAR_IN_OUT
		stOrientation	:	TcVnRotatedRectangle;	(* Resulting rotated rectangle, containig center of mass, lenghts of axes, and rotation angle of the contour in clockwise direction. *)
	END_VAR
	VAR_INPUT
		hrPrev	:	HRESULT;	(* HRESULT indicating the result of previous operations (If SUCCEEDED(hrPrev) equals false, no operation is executed.) *)
	END_VAR

END_FUNCTION

// Functions/Contour Analysis/F_VN_ContourOrientationExp

	{attribute 'TcIecLibraryType'}
	{attribute 'external_name' := 'F_VN_ContourOrientationExp_GUID_6D9A5CB8_D951_2515_7659_68E429EE675D'}
	(* Calculate the orientation of a contour or a set of points. (expert function) *)
	FUNCTION F_VN_ContourOrientationExp : HRESULT
	VAR_INPUT
		ipContour	:	ITcVnContainer;	(* Source point set (ContainerType_Vector_TcVnPoint2_DINT, ContainerType_Vector_TcVnPoint2_REAL, or ContainerType_Vector_TcVnPoint2_LREAL. The elements of this container are the individual points.) *)
	END_VAR
	VAR_IN_OUT
		stOrientation	:	TcVnRotatedRectangle;	(* Resulting rotated rectangle, containig center of mass, lenghts of axes, and rotation angle of the contour in clockwise direction. *)
	END_VAR
	VAR_INPUT
		eMethod	:	ETcVnOrientationMethod;	(* Method for calculating the orientation.  *)
		hrPrev	:	HRESULT;	(* HRESULT indicating the result of previous operations (If SUCCEEDED(hrPrev) equals false, no operation is executed.) *)
	END_VAR

END_FUNCTION

// Functions/Contour Analysis/F_VN_ContourPerimeter

	{attribute 'TcIecLibraryType'}
	{attribute 'external_name' := 'F_VN_ContourPerimeter_GUID_FD268CDC_FBA0_2128_6B0E_1259085DD1F2'}
	(* Computes the perimeter of a contour (curve length if the contour is not closed). *)
	FUNCTION F_VN_ContourPerimeter : HRESULT
	VAR_INPUT
		ipContour	:	ITcVnContainer;	(* Single contour (ContainerType_Vector_TcVnPoint2_DINT or ContainerType_Vector_TcVnPoint2_REAL; The elements of this container are the points of the contour.) *)
	END_VAR
	VAR_IN_OUT
		fPerimeter	:	LREAL;	(* Returns the perimeter of the contour *)
	END_VAR
	VAR_INPUT
		bClosed	:	BOOL;	(* Specifys, if the contour is closed (first and last points connected) or not *)
		hrPrev	:	HRESULT;	(* HRESULT indicating the result of previous operations (If SUCCEEDED(hrPrev) equals false, no operation is executed.) *)
	END_VAR

END_FUNCTION

// Functions/Contour Analysis/F_VN_ContourRoundness

	{attribute 'TcIecLibraryType'}
	{attribute 'external_name' := 'F_VN_ContourRoundness_GUID_3E55BD38_69F7_2890_7527_9BDEF47F5985'}
	(* Computes the roundness of a contour (perimeter^2 / area). *)
	FUNCTION F_VN_ContourRoundness : HRESULT
	VAR_INPUT
		ipContour	:	ITcVnContainer;	(* Single contour (ContainerType_Vector_TcVnPoint2_DINT or ContainerType_Vector_TcVnPoint2_REAL; The elements of this container are the points of the contour.) *)
	END_VAR
	VAR_IN_OUT
		fRoundness	:	LREAL;	(* Returns the roundness of the contour *)
	END_VAR
	VAR_INPUT
		hrPrev	:	HRESULT;	(* HRESULT indicating the result of previous operations (If SUCCEEDED(hrPrev) equals false, no operation is executed.) *)
	END_VAR

END_FUNCTION

// Functions/Contour Analysis/F_VN_ConvexHullPoints

